Fanuc TP program (LS listing): 190220_hosenrohr_oV.ls

/PROG  190220_hosenrohr_oV
/ATTR
COMMENT	= "19-02-22 10:03:29";
PROG_SIZE	= 0;
DEFAULT_GROUP	= 1, 1, *, *, *;
/APPL
    ARC Welding Equipment: 1, *, *, *, *;
/MN
   1:  CALL HOME_ALL;
   1:  UFRAME_NUM = 1;
   1:  UTOOL_NUM = 3;
   1:  COL GUARD ADJUST 150;
   1:  ! -- Layer/Ebene 1 -- !;
   1:  PR[91] = PR[90];
   1:  PR[GP1:91,1] = PR[GP1:90,1] + -0.454;
   1:  PR[GP1:91,2] = PR[GP1:90,2] + 0.328;
   1:  PR[GP1:91,3] = PR[GP1:90,3] + 0.915;
   1:  !Sicherheitspunkt!;
   1:  PR[92] = PR[91];
   1:  PR[92] = PR[GP1:92,3] + 50;
   1:J PR[92];
   1:  !Schweissanfang anfahren!;
   1:L PR[91] R[100]mm/sec CNT100;
   1:  CALL LASER_DRAHT_START;
   1:  PR[GP1:91,1] = PR[GP1:90,1] + -4.023;
   1:  PR[GP1:91,2] = PR[GP1:90,2] + 1.652;
   1:L PR[91] R[100]mm/sec CNT100;
   1:  PR[GP1:91,1] = PR[GP1:90,1] + -5.839;
   1:  PR[GP1:91,2] = PR[GP1:90,2] + 4.932;
   1:L PR[91] R[100]mm/sec CNT100;
   1:  PR[GP1:91,1] = PR[GP1:90,1] + -9.924;
   1:  PR[GP1:91,2] = PR[GP1:90,2] + 16.574;
   1:L PR[91] R[100]mm/sec CNT100;
   1:  PR[GP1:91,1] = PR[GP1:90,1] + -10.007;
   1:  PR[GP1:91,2] = PR[GP1:90,2] + 16.909;
   1:L PR[91] R[100]mm/sec CNT100;
   1:  PR[GP1:91,1] = PR[GP1:90,1] + -10.104;
   1:  PR[GP1:91,2] = PR[GP1:90,2] + 17.121;
   1:L PR[91] R[100]mm/sec CNT100;
   1:  PR[GP1:91,1] = PR[GP1:90,1] + -18.076;
   1:  PR[GP1:91,2] = PR[GP1:90,2] + 26.372;
   1:L PR[91] R[100]mm/sec CNT100;
   1:  PR[GP1:91,1] = PR[GP1:90,1] + -18.276;
   1:  PR[GP1:91,2] = PR[GP1:90,2] + 26.653;
   1:L PR[91] R[100]mm/sec CNT100;
   1:  PR[GP1:91,1] = PR[GP1:90,1] + -18.444;
   1:  PR[GP1:91,2] = PR[GP1:90,2] + 26.815;
   1:L PR[91] R[100]mm/sec CNT100;
   1:  PR[GP1:91,1] = PR[GP1:90,1] + -29.237;
   1:  PR[GP1:91,2] = PR[GP1:90,2] + 32.512;
   1:L PR[91] R[100]mm/sec CNT100;
   1:  PR[GP1:91,1] = PR[GP1:90,1] + -29.526;
   1:  PR[GP1:91,2] = PR[GP1:90,2] + 32.701;
   1:L PR[91] R[100]mm/sec CNT100;
   1:  PR[GP1:91,1] = PR[GP1:90,1] + -29.741;
   1:  PR[GP1:91,2] = PR[GP1:90,2] + 32.790;
   1:L PR[91] R[100]mm/sec CNT100;
   1:  PR[GP1:91,1] = PR[GP1:90,1] + -41.876;
   1:  PR[GP1:91,2] = PR[GP1:90,2] + 34.153;
   1:L PR[91] R[100]mm/sec CNT100;
   1:  PR[GP1:91,1] = PR[GP1:90,1] + -42.214;
   1:  PR[GP1:91,2] = PR[GP1:90,2] + 34.223;
   1:L PR[91] R[100]mm/sec CNT100;
   1:  PR[GP1:91,1] = PR[GP1:90,1] + -42.447;
   1:  PR[GP1:91,2] = PR[GP1:90,2] + 34.227;
   1:L PR[91] R[100]mm/sec CNT100;
   1:  PR[GP1:91,1] = PR[GP1:90,1] + -54.241;
   1:  PR[GP1:91,2] = PR[GP1:90,2] + 31.064;
   1:L PR[91] R[100]mm/sec CNT100;
   1:  PR[GP1:91,1] = PR[GP1:90,1] + -54.581;
   1:  PR[GP1:91,2] = PR[GP1:90,2] + 31.006;
   1:L PR[91] R[100]mm/sec CNT100;
   1:  PR[GP1:91,1] = PR[GP1:90,1] + -54.799;
   1:  PR[GP1:91,2] = PR[GP1:90,2] + 30.925;
   1:L PR[91] R[100]mm/sec CNT100;
   1:  PR[GP1:91,1] = PR[GP1:90,1] + -64.619;
   1:  PR[GP1:91,2] = PR[GP1:90,2] + 23.675;
   1:L PR[91] R[100]mm/sec CNT100;
   1:  PR[GP1:91,1] = PR[GP1:90,1] + -64.915;
   1:  PR[GP1:91,2] = PR[GP1:90,2] + 23.497;
   1:L PR[91] R[100]mm/sec CNT100;
   1:  PR[GP1:91,1] = PR[GP1:90,1] + -65.088;
   1:  PR[GP1:91,2] = PR[GP1:90,2] + 23.342;
   1:L PR[91] R[100]mm/sec CNT100;
   1:  PR[GP1:91,1] = PR[GP1:90,1] + -71.586;
   1:  PR[GP1:91,2] = PR[GP1:90,2] + 12.999;
   1:L PR[91] R[100]mm/sec CNT100;
   1:  PR[GP1:91,1] = PR[GP1:90,1] + -71.796;
   1:  PR[GP1:91,2] = PR[GP1:90,2] + 12.725;
   1:L PR[91] R[100]mm/sec CNT100;
   1:  PR[GP1:91,1] = PR[GP1:90,1] + -71.901;
   1:  PR[GP1:91,2] = PR[GP1:90,2] + 12.518;
   1:L PR[91] R[100]mm/sec CNT100;
   1:  PR[GP1:91,1] = PR[GP1:90,1] + -74.171;
   1:  PR[GP1:91,2] = PR[GP1:90,2] + 0.520;
   1:L PR[91] R[100]mm/sec CNT100;
   1:  PR[GP1:91,1] = PR[GP1:90,1] + -74.266;
   1:  PR[GP1:91,2] = PR[GP1:90,2] + 0.188;
   1:L PR[91] R[100]mm/sec CNT100;
   1:  PR[GP1:91,1] = PR[GP1:90,1] + -74.288;
   1:  PR[GP1:91,2] = PR[GP1:90,2] + -0.044;
   1:L PR[91] R[100]mm/sec CNT100;
   1:  PR[GP1:91,1] = PR[GP1:90,1] + -72.018;
   1:  PR[GP1:91,2] = PR[GP1:90,2] + -12.041;
   1:L PR[91] R[100]mm/sec CNT100;
   1:  PR[GP1:91,1] = PR[GP1:90,1] + -71.986;
   1:  PR[GP1:91,2] = PR[GP1:90,2] + -12.385;
   1:L PR[91] R[100]mm/sec CNT100;
   1:  PR[GP1:91,1] = PR[GP1:90,1] + -71.914;
   1:  PR[GP1:91,2] = PR[GP1:90,2] + -12.636;
   1:L PR[91] R[100]mm/sec CNT100;
   1:  PR[GP1:91,1] = PR[GP1:90,1] + -71.783;
   1:  PR[GP1:91,2] = PR[GP1:90,2] + -12.894;
   1:L PR[91] R[100]mm/sec CNT100;
   1:  PR[GP1:91,1] = PR[GP1:90,1] + -65.286;
   1:  PR[GP1:91,2] = PR[GP1:90,2] + -23.237;
   1:L PR[91] R[100]mm/sec CNT100;
   1:  PR[GP1:91,1] = PR[GP1:90,1] + -65.109;
   1:  PR[GP1:91,2] = PR[GP1:90,2] + -23.467;
   1:L PR[91] R[100]mm/sec CNT100;
   1:  PR[GP1:91,1] = PR[GP1:90,1] + -64.894;
   1:  PR[GP1:91,2] = PR[GP1:90,2] + -23.659;
   1:L PR[91] R[100]mm/sec CNT100;
   1:  PR[GP1:91,1] = PR[GP1:90,1] + -55.074;
   1:  PR[GP1:91,2] = PR[GP1:90,2] + -30.910;
   1:L PR[91] R[100]mm/sec CNT100;
   1:  PR[GP1:91,1] = PR[GP1:90,1] + -54.826;
   1:  PR[GP1:91,2] = PR[GP1:90,2] + -31.059;
   1:L PR[91] R[100]mm/sec CNT100;
   1:  PR[GP1:91,1] = PR[GP1:90,1] + -54.555;
   1:  PR[GP1:91,2] = PR[GP1:90,2] + -31.160;
   1:L PR[91] R[100]mm/sec CNT100;
   1:  PR[GP1:91,1] = PR[GP1:90,1] + -42.760;
   1:  PR[GP1:91,2] = PR[GP1:90,2] + -34.323;
   1:L PR[91] R[100]mm/sec CNT100;
   1:  PR[GP1:91,1] = PR[GP1:90,1] + -42.475;
   1:  PR[GP1:91,2] = PR[GP1:90,2] + -34.372;
   1:L PR[91] R[100]mm/sec CNT100;
   1:  PR[GP1:91,1] = PR[GP1:90,1] + -42.186;
   1:  PR[GP1:91,2] = PR[GP1:90,2] + -34.367;
   1:L PR[91] R[100]mm/sec CNT100;
   1:  PR[GP1:91,1] = PR[GP1:90,1] + -30.051;
   1:  PR[GP1:91,2] = PR[GP1:90,2] + -33.004;
   1:L PR[91] R[100]mm/sec CNT100;
   1:  PR[GP1:91,1] = PR[GP1:90,1] + -29.768;
   1:  PR[GP1:91,2] = PR[GP1:90,2] + -32.945;
   1:L PR[91] R[100]mm/sec CNT100;
   1:  PR[GP1:91,1] = PR[GP1:90,1] + -29.500;
   1:  PR[GP1:91,2] = PR[GP1:90,2] + -32.835;
   1:L PR[91] R[100]mm/sec CNT100;
   1:  PR[GP1:91,1] = PR[GP1:90,1] + -18.706;
   1:  PR[GP1:91,2] = PR[GP1:90,2] + -27.137;
   1:L PR[91] R[100]mm/sec CNT100;
   1:  PR[GP1:91,1] = PR[GP1:90,1] + -18.464;
   1:  PR[GP1:91,2] = PR[GP1:90,2] + -26.978;
   1:L PR[91] R[100]mm/sec CNT100;
   1:  PR[GP1:91,1] = PR[GP1:90,1] + -18.256;
   1:  PR[GP1:91,2] = PR[GP1:90,2] + -26.778;
   1:L PR[91] R[100]mm/sec CNT100;
   1:  PR[GP1:91,1] = PR[GP1:90,1] + -10.284;
   1:  PR[GP1:91,2] = PR[GP1:90,2] + -17.526;
   1:L PR[91] R[100]mm/sec CNT100;
   1:  PR[GP1:91,1] = PR[GP1:90,1] + -10.116;
   1:  PR[GP1:91,2] = PR[GP1:90,2] + -17.290;
   1:L PR[91] R[100]mm/sec CNT100;
   1:  PR[GP1:91,1] = PR[GP1:90,1] + -9.995;
   1:  PR[GP1:91,2] = PR[GP1:90,2] + -17.028;
   1:L PR[91] R[100]mm/sec CNT100;
   1:  PR[GP1:91,1] = PR[GP1:90,1] + -5.955;
   1:  PR[GP1:91,2] = PR[GP1:90,2] + -5.512;
   1:L PR[91] R[100]mm/sec CNT100;
   1:  PR[GP1:91,1] = PR[GP1:90,1] + -5.853;
   1:  PR[GP1:91,2] = PR[GP1:90,2] + -5.100;
   1:L PR[91] R[100]mm/sec CNT100;
   1:  PR[GP1:91,1] = PR[GP1:90,1] + -4.023;
   1:  PR[GP1:91,2] = PR[GP1:90,2] + -1.796;
   1:L PR[91] R[100]mm/sec CNT100;
   1:  PR[GP1:91,1] = PR[GP1:90,1] + -0.454;
   1:  PR[GP1:91,2] = PR[GP1:90,2] + -0.472;
   1:L PR[91] R[100]mm/sec CNT100;
   1:  PR[GP1:91,1] = PR[GP1:90,1] + 0.667;
   1:L PR[91] R[100]mm/sec CNT100;
   1:  PR[GP1:91,1] = PR[GP1:90,1] + 4.237;
   1:  PR[GP1:91,2] = PR[GP1:90,2] + -1.796;
   1:L PR[91] R[100]mm/sec CNT100;
   1:  PR[GP1:91,1] = PR[GP1:90,1] + 6.052;
   1:  PR[GP1:91,2] = PR[GP1:90,2] + -5.076;
   1:L PR[91] R[100]mm/sec CNT100;
   1:  PR[GP1:91,1] = PR[GP1:90,1] + 10.137;
   1:  PR[GP1:91,2] = PR[GP1:90,2] + -16.718;
   1:L PR[91] R[100]mm/sec CNT100;
   1:  PR[GP1:91,1] = PR[GP1:90,1] + 10.221;
   1:  PR[GP1:91,2] = PR[GP1:90,2] + -17.053;
   1:L PR[91] R[100]mm/sec CNT100;
   1:  PR[GP1:91,1] = PR[GP1:90,1] + 10.318;
   1:  PR[GP1:91,2] = PR[GP1:90,2] + -17.265;
   1:L PR[91] R[100]mm/sec CNT100;
   1:  PR[GP1:91,1] = PR[GP1:90,1] + 18.289;
   1:  PR[GP1:91,2] = PR[GP1:90,2] + -26.516;
   1:L PR[91] R[100]mm/sec CNT100;
   1:  PR[GP1:91,1] = PR[GP1:90,1] + 18.489;
   1:  PR[GP1:91,2] = PR[GP1:90,2] + -26.797;
   1:L PR[91] R[100]mm/sec CNT100;
   1:  PR[GP1:91,1] = PR[GP1:90,1] + 18.657;
   1:  PR[GP1:91,2] = PR[GP1:90,2] + -26.959;
   1:L PR[91] R[100]mm/sec CNT100;
   1:  PR[GP1:91,1] = PR[GP1:90,1] + 29.451;
   1:  PR[GP1:91,2] = PR[GP1:90,2] + -32.656;
   1:L PR[91] R[100]mm/sec CNT100;
   1:  PR[GP1:91,1] = PR[GP1:90,1] + 29.740;
   1:  PR[GP1:91,2] = PR[GP1:90,2] + -32.845;
   1:L PR[91] R[100]mm/sec CNT100;
   1:  PR[GP1:91,1] = PR[GP1:90,1] + 29.955;
   1:  PR[GP1:91,2] = PR[GP1:90,2] + -32.934;
   1:L PR[91] R[100]mm/sec CNT100;
   1:  PR[GP1:91,1] = PR[GP1:90,1] + 42.089;
   1:  PR[GP1:91,2] = PR[GP1:90,2] + -34.297;
   1:L PR[91] R[100]mm/sec CNT100;
   1:  PR[GP1:91,1] = PR[GP1:90,1] + 42.427;
   1:  PR[GP1:91,2] = PR[GP1:90,2] + -34.367;
   1:L PR[91] R[100]mm/sec CNT100;
   1:  PR[GP1:91,1] = PR[GP1:90,1] + 42.660;
   1:  PR[GP1:91,2] = PR[GP1:90,2] + -34.371;
   1:L PR[91] R[100]mm/sec CNT100;
   1:  PR[GP1:91,1] = PR[GP1:90,1] + 54.454;
   1:  PR[GP1:91,2] = PR[GP1:90,2] + -31.208;
   1:L PR[91] R[100]mm/sec CNT100;
   1:  PR[GP1:91,1] = PR[GP1:90,1] + 54.794;
   1:  PR[GP1:91,2] = PR[GP1:90,2] + -31.150;
   1:L PR[91] R[100]mm/sec CNT100;
   1:  PR[GP1:91,1] = PR[GP1:90,1] + 55.013;
   1:  PR[GP1:91,2] = PR[GP1:90,2] + -31.069;
   1:L PR[91] R[100]mm/sec CNT100;
   1:  PR[GP1:91,1] = PR[GP1:90,1] + 64.832;
   1:  PR[GP1:91,2] = PR[GP1:90,2] + -23.819;
   1:L PR[91] R[100]mm/sec CNT100;
   1:  PR[GP1:91,1] = PR[GP1:90,1] + 65.128;
   1:  PR[GP1:91,2] = PR[GP1:90,2] + -23.641;
   1:L PR[91] R[100]mm/sec CNT100;
   1:  PR[GP1:91,1] = PR[GP1:90,1] + 65.302;
   1:  PR[GP1:91,2] = PR[GP1:90,2] + -23.486;
   1:L PR[91] R[100]mm/sec CNT100;
   1:  PR[GP1:91,1] = PR[GP1:90,1] + 71.799;
   1:  PR[GP1:91,2] = PR[GP1:90,2] + -13.143;
   1:L PR[91] R[100]mm/sec CNT100;
   1:  PR[GP1:91,1] = PR[GP1:90,1] + 72.009;
   1:  PR[GP1:91,2] = PR[GP1:90,2] + -12.869;
   1:L PR[91] R[100]mm/sec CNT100;
   1:  PR[GP1:91,1] = PR[GP1:90,1] + 72.114;
   1:  PR[GP1:91,2] = PR[GP1:90,2] + -12.661;
   1:L PR[91] R[100]mm/sec CNT100;
   1:  PR[GP1:91,1] = PR[GP1:90,1] + 74.384;
   1:  PR[GP1:91,2] = PR[GP1:90,2] + -0.664;
   1:L PR[91] R[100]mm/sec CNT100;
   1:  PR[GP1:91,1] = PR[GP1:90,1] + 74.480;
   1:  PR[GP1:91,2] = PR[GP1:90,2] + -0.332;
   1:L PR[91] R[100]mm/sec CNT100;
   1:  PR[GP1:91,1] = PR[GP1:90,1] + 74.501;
   1:  PR[GP1:91,2] = PR[GP1:90,2] + -0.100;
   1:L PR[91] R[100]mm/sec CNT100;
   1:  PR[GP1:91,1] = PR[GP1:90,1] + 72.231;
   1:  PR[GP1:91,2] = PR[GP1:90,2] + 11.897;
   1:L PR[91] R[100]mm/sec CNT100;
   1:  PR[GP1:91,1] = PR[GP1:90,1] + 72.199;
   1:  PR[GP1:91,2] = PR[GP1:90,2] + 12.241;
   1:L PR[91] R[100]mm/sec CNT100;
   1:  PR[GP1:91,1] = PR[GP1:90,1] + 72.127;
   1:  PR[GP1:91,2] = PR[GP1:90,2] + 12.492;
   1:L PR[91] R[100]mm/sec CNT100;
   1:  PR[GP1:91,1] = PR[GP1:90,1] + 71.996;
   1:  PR[GP1:91,2] = PR[GP1:90,2] + 12.750;
   1:L PR[91] R[100]mm/sec CNT100;
   1:  PR[GP1:91,1] = PR[GP1:90,1] + 65.499;
   1:  PR[GP1:91,2] = PR[GP1:90,2] + 23.093;
   1:L PR[91] R[100]mm/sec CNT100;
   1:  PR[GP1:91,1] = PR[GP1:90,1] + 65.323;
   1:  PR[GP1:91,2] = PR[GP1:90,2] + 23.323;
   1:L PR[91] R[100]mm/sec CNT100;
   1:  PR[GP1:91,1] = PR[GP1:90,1] + 65.107;
   1:  PR[GP1:91,2] = PR[GP1:90,2] + 23.515;
   1:L PR[91] R[100]mm/sec CNT100;
   1:  PR[GP1:91,1] = PR[GP1:90,1] + 55.287;
   1:  PR[GP1:91,2] = PR[GP1:90,2] + 30.766;
   1:L PR[91] R[100]mm/sec CNT100;
   1:  PR[GP1:91,1] = PR[GP1:90,1] + 55.039;
   1:  PR[GP1:91,2] = PR[GP1:90,2] + 30.915;
   1:L PR[91] R[100]mm/sec CNT100;
   1:  PR[GP1:91,1] = PR[GP1:90,1] + 54.768;
   1:  PR[GP1:91,2] = PR[GP1:90,2] + 31.016;
   1:L PR[91] R[100]mm/sec CNT100;
   1:  PR[GP1:91,1] = PR[GP1:90,1] + 42.973;
   1:  PR[GP1:91,2] = PR[GP1:90,2] + 34.179;
   1:L PR[91] R[100]mm/sec CNT100;
   1:  PR[GP1:91,1] = PR[GP1:90,1] + 42.688;
   1:  PR[GP1:91,2] = PR[GP1:90,2] + 34.228;
   1:L PR[91] R[100]mm/sec CNT100;
   1:  PR[GP1:91,1] = PR[GP1:90,1] + 42.399;
   1:  PR[GP1:91,2] = PR[GP1:90,2] + 34.223;
   1:L PR[91] R[100]mm/sec CNT100;
   1:  PR[GP1:91,1] = PR[GP1:90,1] + 30.264;
   1:  PR[GP1:91,2] = PR[GP1:90,2] + 32.860;
   1:L PR[91] R[100]mm/sec CNT100;
   1:  PR[GP1:91,1] = PR[GP1:90,1] + 29.981;
   1:  PR[GP1:91,2] = PR[GP1:90,2] + 32.801;
   1:L PR[91] R[100]mm/sec CNT100;
   1:  PR[GP1:91,1] = PR[GP1:90,1] + 29.714;
   1:  PR[GP1:91,2] = PR[GP1:90,2] + 32.691;
   1:L PR[91] R[100]mm/sec CNT100;
   1:  PR[GP1:91,1] = PR[GP1:90,1] + 18.920;
   1:  PR[GP1:91,2] = PR[GP1:90,2] + 26.993;
   1:L PR[91] R[100]mm/sec CNT100;
   1:  PR[GP1:91,1] = PR[GP1:90,1] + 18.678;
   1:  PR[GP1:91,2] = PR[GP1:90,2] + 26.834;
   1:L PR[91] R[100]mm/sec CNT100;
   1:  PR[GP1:91,1] = PR[GP1:90,1] + 18.469;
   1:  PR[GP1:91,2] = PR[GP1:90,2] + 26.634;
   1:L PR[91] R[100]mm/sec CNT100;
   1:  PR[GP1:91,1] = PR[GP1:90,1] + 10.497;
   1:  PR[GP1:91,2] = PR[GP1:90,2] + 17.382;
   1:L PR[91] R[100]mm/sec CNT100;
   1:  PR[GP1:91,1] = PR[GP1:90,1] + 10.330;
   1:  PR[GP1:91,2] = PR[GP1:90,2] + 17.146;
   1:L PR[91] R[100]mm/sec CNT100;
   1:  PR[GP1:91,1] = PR[GP1:90,1] + 10.209;
   1:  PR[GP1:91,2] = PR[GP1:90,2] + 16.884;
   1:L PR[91] R[100]mm/sec CNT100;
   1:  PR[GP1:91,1] = PR[GP1:90,1] + 6.168;
   1:  PR[GP1:91,2] = PR[GP1:90,2] + 5.368;
   1:L PR[91] R[100]mm/sec CNT100;
   1:  PR[GP1:91,1] = PR[GP1:90,1] + 6.066;
   1:  PR[GP1:91,2] = PR[GP1:90,2] + 4.956;
   1:L PR[91] R[100]mm/sec CNT100;
   1:  PR[GP1:91,1] = PR[GP1:90,1] + 4.237;
   1:  PR[GP1:91,2] = PR[GP1:90,2] + 1.652;
   1:L PR[91] R[100]mm/sec CNT100;
   1:  PR[GP1:91,1] = PR[GP1:90,1] + 0.667;
   1:  PR[GP1:91,2] = PR[GP1:90,2] + 0.328;
   1:L PR[91] R[100]mm/sec CNT100;
   1:  PR[GP1:91,1] = PR[GP1:90,1] + -0.454;
   1:L PR[91] R[100]mm/sec CNT100;
   1:  ! -- Layer/Ebene 2 -- !;
   1:  PR[91] = PR[90];
   1:  PR[GP1:91,1] = PR[GP1:90,1] + -4.023;
   1:  PR[GP1:91,2] = PR[GP1:90,2] + 1.652;
   1:  PR[GP1:91,3] = PR[GP1:90,3] + 1.525;
   1:L PR[91] R[100]mm/sec CNT100;
   1:  PR[GP1:91,1] = PR[GP1:90,1] + -5.839;
   1:  PR[GP1:91,2] = PR[GP1:90,2] + 4.932;
   1:L PR[91] R[100]mm/sec CNT100;
   1:  PR[GP1:91,1] = PR[GP1:90,1] + -9.513;
   1:  PR[GP1:91,2] = PR[GP1:90,2] + 15.405;
   1:L PR[91] R[100]mm/sec CNT100;
   1:  PR[GP1:91,1] = PR[GP1:90,1] + -9.747;
   1:  PR[GP1:91,2] = PR[GP1:90,2] + 16.344;
   1:L PR[91] R[100]mm/sec CNT100;
   1:  PR[GP1:91,1] = PR[GP1:90,1] + -10.105;
   1:  PR[GP1:91,2] = PR[GP1:90,2] + 17.121;
   1:L PR[91] R[100]mm/sec CNT100;
   1:  PR[GP1:91,1] = PR[GP1:90,1] + -17.267;
   1:  PR[GP1:91,2] = PR[GP1:90,2] + 25.433;
   1:L PR[91] R[100]mm/sec CNT100;
   1:  PR[GP1:91,1] = PR[GP1:90,1] + -17.828;
   1:  PR[GP1:91,2] = PR[GP1:90,2] + 26.222;
   1:L PR[91] R[100]mm/sec CNT100;
   1:  PR[GP1:91,1] = PR[GP1:90,1] + -18.444;
   1:  PR[GP1:91,2] = PR[GP1:90,2] + 26.815;
   1:L PR[91] R[100]mm/sec CNT100;
   1:  PR[GP1:91,1] = PR[GP1:90,1] + -28.141;
   1:  PR[GP1:91,2] = PR[GP1:90,2] + 31.934;
   1:L PR[91] R[100]mm/sec CNT100;
   1:  PR[GP1:91,1] = PR[GP1:90,1] + -28.952;
   1:  PR[GP1:91,2] = PR[GP1:90,2] + 32.464;
   1:L PR[91] R[100]mm/sec CNT100;
   1:  PR[GP1:91,1] = PR[GP1:90,1] + -29.742;
   1:  PR[GP1:91,2] = PR[GP1:90,2] + 32.791;
   1:L PR[91] R[100]mm/sec CNT100;
   1:  PR[GP1:91,1] = PR[GP1:90,1] + -40.644;
   1:  PR[GP1:91,2] = PR[GP1:90,2] + 34.015;
   1:L PR[91] R[100]mm/sec CNT100;
   1:  PR[GP1:91,1] = PR[GP1:90,1] + -41.592;
   1:  PR[GP1:91,2] = PR[GP1:90,2] + 34.212;
   1:L PR[91] R[100]mm/sec CNT100;
   1:  PR[GP1:91,1] = PR[GP1:90,1] + -42.447;
   1:  PR[GP1:91,2] = PR[GP1:90,2] + 34.227;
   1:L PR[91] R[100]mm/sec CNT100;
   1:  PR[GP1:91,1] = PR[GP1:90,1] + -53.043;
   1:  PR[GP1:91,2] = PR[GP1:90,2] + 31.385;
   1:L PR[91] R[100]mm/sec CNT100;
   1:  PR[GP1:91,1] = PR[GP1:90,1] + -53.998;
   1:  PR[GP1:91,2] = PR[GP1:90,2] + 31.223;
   1:L PR[91] R[100]mm/sec CNT100;
   1:  PR[GP1:91,1] = PR[GP1:90,1] + -54.800;
   1:  PR[GP1:91,2] = PR[GP1:90,2] + 30.925;
   1:L PR[91] R[100]mm/sec CNT100;
   1:  PR[GP1:91,1] = PR[GP1:90,1] + -63.622;
   1:  PR[GP1:91,2] = PR[GP1:90,2] + 24.411;
   1:L PR[91] R[100]mm/sec CNT100;
   1:  PR[GP1:91,1] = PR[GP1:90,1] + -64.451;
   1:  PR[GP1:91,2] = PR[GP1:90,2] + 23.911;
   1:L PR[91] R[100]mm/sec CNT100;
   1:  PR[GP1:91,1] = PR[GP1:90,1] + -65.089;
   1:  PR[GP1:91,2] = PR[GP1:90,2] + 23.341;
   1:L PR[91] R[100]mm/sec CNT100;
   1:  PR[GP1:91,1] = PR[GP1:90,1] + -70.926;
   1:  PR[GP1:91,2] = PR[GP1:90,2] + 14.049;
   1:L PR[91] R[100]mm/sec CNT100;
   1:  PR[GP1:91,1] = PR[GP1:90,1] + -71.515;
   1:  PR[GP1:91,2] = PR[GP1:90,2] + 13.281;
   1:L PR[91] R[100]mm/sec CNT100;
   1:  PR[GP1:91,1] = PR[GP1:90,1] + -71.901;
   1:  PR[GP1:91,2] = PR[GP1:90,2] + 12.517;
   1:L PR[91] R[100]mm/sec CNT100;
   1:  PR[GP1:91,1] = PR[GP1:90,1] + -73.940;
   1:  PR[GP1:91,2] = PR[GP1:90,2] + 1.738;
   1:L PR[91] R[100]mm/sec CNT100;
   1:  PR[GP1:91,1] = PR[GP1:90,1] + -74.208;
   1:  PR[GP1:91,2] = PR[GP1:90,2] + 0.808;
   1:L PR[91] R[100]mm/sec CNT100;
   1:  PR[GP1:91,1] = PR[GP1:90,1] + -74.288;
   1:  PR[GP1:91,2] = PR[GP1:90,2] + -0.044;
   1:L PR[91] R[100]mm/sec CNT100;
   1:  PR[GP1:91,1] = PR[GP1:90,1] + -72.249;
   1:  PR[GP1:91,2] = PR[GP1:90,2] + -10.823;
   1:L PR[91] R[100]mm/sec CNT100;
   1:  PR[GP1:91,1] = PR[GP1:90,1] + -72.158;
   1:  PR[GP1:91,2] = PR[GP1:90,2] + -11.787;
   1:L PR[91] R[100]mm/sec CNT100;
   1:  PR[GP1:91,1] = PR[GP1:90,1] + -71.914;
   1:  PR[GP1:91,2] = PR[GP1:90,2] + -12.636;
   1:L PR[91] R[100]mm/sec CNT100;
   1:  PR[GP1:91,1] = PR[GP1:90,1] + -71.503;
   1:  PR[GP1:91,2] = PR[GP1:90,2] + -13.450;
   1:L PR[91] R[100]mm/sec CNT100;
   1:  PR[GP1:91,1] = PR[GP1:90,1] + -65.665;
   1:  PR[GP1:91,2] = PR[GP1:90,2] + -22.742;
   1:L PR[91] R[100]mm/sec CNT100;
   1:  PR[GP1:91,1] = PR[GP1:90,1] + -65.110;
   1:  PR[GP1:91,2] = PR[GP1:90,2] + -23.466;
   1:L PR[91] R[100]mm/sec CNT100;
   1:  PR[GP1:91,1] = PR[GP1:90,1] + -64.430;
   1:  PR[GP1:91,2] = PR[GP1:90,2] + -24.074;
   1:L PR[91] R[100]mm/sec CNT100;
   1:  PR[GP1:91,1] = PR[GP1:90,1] + -55.607;
   1:  PR[GP1:91,2] = PR[GP1:90,2] + -30.588;
   1:L PR[91] R[100]mm/sec CNT100;
   1:  PR[GP1:91,1] = PR[GP1:90,1] + -54.826;
   1:  PR[GP1:91,2] = PR[GP1:90,2] + -31.059;
   1:L PR[91] R[100]mm/sec CNT100;
   1:  PR[GP1:91,1] = PR[GP1:90,1] + -53.971;
   1:  PR[GP1:91,2] = PR[GP1:90,2] + -31.376;
   1:L PR[91] R[100]mm/sec CNT100;
   1:  PR[GP1:91,1] = PR[GP1:90,1] + -43.375;
   1:  PR[GP1:91,2] = PR[GP1:90,2] + -34.219;
   1:L PR[91] R[100]mm/sec CNT100;
   1:  PR[GP1:91,1] = PR[GP1:90,1] + -42.476;
   1:  PR[GP1:91,2] = PR[GP1:90,2] + -34.372;
   1:L PR[91] R[100]mm/sec CNT100;
   1:  PR[GP1:91,1] = PR[GP1:90,1] + -41.564;
   1:  PR[GP1:91,2] = PR[GP1:90,2] + -34.355;
   1:L PR[91] R[100]mm/sec CNT100;
   1:  PR[GP1:91,1] = PR[GP1:90,1] + -30.661;
   1:  PR[GP1:91,2] = PR[GP1:90,2] + -33.131;
   1:L PR[91] R[100]mm/sec CNT100;
   1:  PR[GP1:91,1] = PR[GP1:90,1] + -29.768;
   1:  PR[GP1:91,2] = PR[GP1:90,2] + -32.945;
   1:L PR[91] R[100]mm/sec CNT100;
   1:  PR[GP1:91,1] = PR[GP1:90,1] + -28.926;
   1:  PR[GP1:91,2] = PR[GP1:90,2] + -32.597;
   1:L PR[91] R[100]mm/sec CNT100;
   1:  PR[GP1:91,1] = PR[GP1:90,1] + -19.228;
   1:  PR[GP1:91,2] = PR[GP1:90,2] + -27.478;
   1:L PR[91] R[100]mm/sec CNT100;
   1:  PR[GP1:91,1] = PR[GP1:90,1] + -18.465;
   1:  PR[GP1:91,2] = PR[GP1:90,2] + -26.979;
   1:L PR[91] R[100]mm/sec CNT100;
   1:  PR[GP1:91,1] = PR[GP1:90,1] + -17.807;
   1:  PR[GP1:91,2] = PR[GP1:90,2] + -26.346;
   1:L PR[91] R[100]mm/sec CNT100;
   1:  PR[GP1:91,1] = PR[GP1:90,1] + -10.645;
   1:  PR[GP1:91,2] = PR[GP1:90,2] + -18.034;
   1:L PR[91] R[100]mm/sec CNT100;
   1:  PR[GP1:91,1] = PR[GP1:90,1] + -10.117;
   1:  PR[GP1:91,2] = PR[GP1:90,2] + -17.291;
   1:L PR[91] R[100]mm/sec CNT100;
   1:  PR[GP1:91,1] = PR[GP1:90,1] + -9.736;
   1:  PR[GP1:91,2] = PR[GP1:90,2] + -16.462;
   1:L PR[91] R[100]mm/sec CNT100;
   1:  PR[GP1:91,1] = PR[GP1:90,1] + -6.106;
   1:  PR[GP1:91,2] = PR[GP1:90,2] + -6.117;
   1:L PR[91] R[100]mm/sec CNT100;
   1:  PR[GP1:91,1] = PR[GP1:90,1] + -5.853;
   1:  PR[GP1:91,2] = PR[GP1:90,2] + -5.100;
   1:L PR[91] R[100]mm/sec CNT100;
   1:  PR[GP1:91,1] = PR[GP1:90,1] + -4.023;
   1:  PR[GP1:91,2] = PR[GP1:90,2] + -1.796;
   1:L PR[91] R[100]mm/sec CNT100;
   1:  PR[GP1:91,1] = PR[GP1:90,1] + -0.454;
   1:  PR[GP1:91,2] = PR[GP1:90,2] + -0.472;
   1:L PR[91] R[100]mm/sec CNT100;
   1:  PR[GP1:91,1] = PR[GP1:90,1] + 0.667;
   1:L PR[91] R[100]mm/sec CNT100;
   1:  PR[GP1:91,1] = PR[GP1:90,1] + 4.237;
   1:  PR[GP1:91,2] = PR[GP1:90,2] + -1.796;
   1:L PR[91] R[100]mm/sec CNT100;
   1:  PR[GP1:91,1] = PR[GP1:90,1] + 6.052;
   1:  PR[GP1:91,2] = PR[GP1:90,2] + -5.076;
   1:L PR[91] R[100]mm/sec CNT100;
   1:  PR[GP1:91,1] = PR[GP1:90,1] + 9.727;
   1:  PR[GP1:91,2] = PR[GP1:90,2] + -15.549;
   1:L PR[91] R[100]mm/sec CNT100;
   1:  PR[GP1:91,1] = PR[GP1:90,1] + 9.961;
   1:  PR[GP1:91,2] = PR[GP1:90,2] + -16.488;
   1:L PR[91] R[100]mm/sec CNT100;
   1:  PR[GP1:91,1] = PR[GP1:90,1] + 10.318;
   1:  PR[GP1:91,2] = PR[GP1:90,2] + -17.265;
   1:L PR[91] R[100]mm/sec CNT100;
   1:  PR[GP1:91,1] = PR[GP1:90,1] + 17.480;
   1:  PR[GP1:91,2] = PR[GP1:90,2] + -25.577;
   1:L PR[91] R[100]mm/sec CNT100;
   1:  PR[GP1:91,1] = PR[GP1:90,1] + 18.041;
   1:  PR[GP1:91,2] = PR[GP1:90,2] + -26.366;
   1:L PR[91] R[100]mm/sec CNT100;
   1:  PR[GP1:91,1] = PR[GP1:90,1] + 18.657;
   1:  PR[GP1:91,2] = PR[GP1:90,2] + -26.959;
   1:L PR[91] R[100]mm/sec CNT100;
   1:  PR[GP1:91,1] = PR[GP1:90,1] + 28.355;
   1:  PR[GP1:91,2] = PR[GP1:90,2] + -32.078;
   1:L PR[91] R[100]mm/sec CNT100;
   1:  PR[GP1:91,1] = PR[GP1:90,1] + 29.165;
   1:  PR[GP1:91,2] = PR[GP1:90,2] + -32.608;
   1:L PR[91] R[100]mm/sec CNT100;
   1:  PR[GP1:91,1] = PR[GP1:90,1] + 29.955;
   1:  PR[GP1:91,2] = PR[GP1:90,2] + -32.934;
   1:L PR[91] R[100]mm/sec CNT100;
   1:  PR[GP1:91,1] = PR[GP1:90,1] + 40.857;
   1:  PR[GP1:91,2] = PR[GP1:90,2] + -34.159;
   1:L PR[91] R[100]mm/sec CNT100;
   1:  PR[GP1:91,1] = PR[GP1:90,1] + 41.805;
   1:  PR[GP1:91,2] = PR[GP1:90,2] + -34.356;
   1:L PR[91] R[100]mm/sec CNT100;
   1:  PR[GP1:91,1] = PR[GP1:90,1] + 42.660;
   1:  PR[GP1:91,2] = PR[GP1:90,2] + -34.371;
   1:L PR[91] R[100]mm/sec CNT100;
   1:  PR[GP1:91,1] = PR[GP1:90,1] + 53.257;
   1:  PR[GP1:91,2] = PR[GP1:90,2] + -31.529;
   1:L PR[91] R[100]mm/sec CNT100;
   1:  PR[GP1:91,1] = PR[GP1:90,1] + 54.211;
   1:  PR[GP1:91,2] = PR[GP1:90,2] + -31.367;
   1:L PR[91] R[100]mm/sec CNT100;
   1:  PR[GP1:91,1] = PR[GP1:90,1] + 55.013;
   1:  PR[GP1:91,2] = PR[GP1:90,2] + -31.069;
   1:L PR[91] R[100]mm/sec CNT100;
   1:  PR[GP1:91,1] = PR[GP1:90,1] + 63.835;
   1:  PR[GP1:91,2] = PR[GP1:90,2] + -24.555;
   1:L PR[91] R[100]mm/sec CNT100;
   1:  PR[GP1:91,1] = PR[GP1:90,1] + 64.664;
   1:  PR[GP1:91,2] = PR[GP1:90,2] + -24.055;
   1:L PR[91] R[100]mm/sec CNT100;
   1:  PR[GP1:91,1] = PR[GP1:90,1] + 65.302;
   1:  PR[GP1:91,2] = PR[GP1:90,2] + -23.485;
   1:L PR[91] R[100]mm/sec CNT100;
   1:  PR[GP1:91,1] = PR[GP1:90,1] + 71.140;
   1:  PR[GP1:91,2] = PR[GP1:90,2] + -14.193;
   1:L PR[91] R[100]mm/sec CNT100;
   1:  PR[GP1:91,1] = PR[GP1:90,1] + 71.729;
   1:  PR[GP1:91,2] = PR[GP1:90,2] + -13.425;
   1:L PR[91] R[100]mm/sec CNT100;
   1:  PR[GP1:91,1] = PR[GP1:90,1] + 72.114;
   1:  PR[GP1:91,2] = PR[GP1:90,2] + -12.661;
   1:L PR[91] R[100]mm/sec CNT100;
   1:  PR[GP1:91,1] = PR[GP1:90,1] + 74.154;
   1:  PR[GP1:91,2] = PR[GP1:90,2] + -1.882;
   1:L PR[91] R[100]mm/sec CNT100;
   1:  PR[GP1:91,1] = PR[GP1:90,1] + 74.421;
   1:  PR[GP1:91,2] = PR[GP1:90,2] + -0.952;
   1:L PR[91] R[100]mm/sec CNT100;
   1:  PR[GP1:91,1] = PR[GP1:90,1] + 74.501;
   1:  PR[GP1:91,2] = PR[GP1:90,2] + -0.100;
   1:L PR[91] R[100]mm/sec CNT100;
   1:  PR[GP1:91,1] = PR[GP1:90,1] + 72.462;
   1:  PR[GP1:91,2] = PR[GP1:90,2] + 10.679;
   1:L PR[91] R[100]mm/sec CNT100;
   1:  PR[GP1:91,1] = PR[GP1:90,1] + 72.371;
   1:  PR[GP1:91,2] = PR[GP1:90,2] + 11.643;
   1:L PR[91] R[100]mm/sec CNT100;
   1:  PR[GP1:91,1] = PR[GP1:90,1] + 72.127;
   1:  PR[GP1:91,2] = PR[GP1:90,2] + 12.492;
   1:L PR[91] R[100]mm/sec CNT100;
   1:  PR[GP1:91,1] = PR[GP1:90,1] + 71.716;
   1:  PR[GP1:91,2] = PR[GP1:90,2] + 13.306;
   1:L PR[91] R[100]mm/sec CNT100;
   1:  PR[GP1:91,1] = PR[GP1:90,1] + 65.878;
   1:  PR[GP1:91,2] = PR[GP1:90,2] + 22.599;
   1:L PR[91] R[100]mm/sec CNT100;
   1:  PR[GP1:91,1] = PR[GP1:90,1] + 65.323;
   1:  PR[GP1:91,2] = PR[GP1:90,2] + 23.322;
   1:L PR[91] R[100]mm/sec CNT100;
   1:  PR[GP1:91,1] = PR[GP1:90,1] + 64.643;
   1:  PR[GP1:91,2] = PR[GP1:90,2] + 23.930;
   1:L PR[91] R[100]mm/sec CNT100;
   1:  PR[GP1:91,1] = PR[GP1:90,1] + 55.820;
   1:  PR[GP1:91,2] = PR[GP1:90,2] + 30.444;
   1:L PR[91] R[100]mm/sec CNT100;
   1:  PR[GP1:91,1] = PR[GP1:90,1] + 55.039;
   1:  PR[GP1:91,2] = PR[GP1:90,2] + 30.915;
   1:L PR[91] R[100]mm/sec CNT100;
   1:  PR[GP1:91,1] = PR[GP1:90,1] + 54.185;
   1:  PR[GP1:91,2] = PR[GP1:90,2] + 31.232;
   1:L PR[91] R[100]mm/sec CNT100;
   1:  PR[GP1:91,1] = PR[GP1:90,1] + 43.588;
   1:  PR[GP1:91,2] = PR[GP1:90,2] + 34.075;
   1:L PR[91] R[100]mm/sec CNT100;
   1:  PR[GP1:91,1] = PR[GP1:90,1] + 42.689;
   1:  PR[GP1:91,2] = PR[GP1:90,2] + 34.228;
   1:L PR[91] R[100]mm/sec CNT100;
   1:  PR[GP1:91,1] = PR[GP1:90,1] + 41.777;
   1:  PR[GP1:91,2] = PR[GP1:90,2] + 34.211;
   1:L PR[91] R[100]mm/sec CNT100;
   1:  PR[GP1:91,1] = PR[GP1:90,1] + 30.875;
   1:  PR[GP1:91,2] = PR[GP1:90,2] + 32.987;
   1:L PR[91] R[100]mm/sec CNT100;
   1:  PR[GP1:91,1] = PR[GP1:90,1] + 29.982;
   1:  PR[GP1:91,2] = PR[GP1:90,2] + 32.801;
   1:L PR[91] R[100]mm/sec CNT100;
   1:  PR[GP1:91,1] = PR[GP1:90,1] + 29.139;
   1:  PR[GP1:91,2] = PR[GP1:90,2] + 32.453;
   1:L PR[91] R[100]mm/sec CNT100;
   1:  PR[GP1:91,1] = PR[GP1:90,1] + 19.441;
   1:  PR[GP1:91,2] = PR[GP1:90,2] + 27.334;
   1:L PR[91] R[100]mm/sec CNT100;
   1:  PR[GP1:91,1] = PR[GP1:90,1] + 18.678;
   1:  PR[GP1:91,2] = PR[GP1:90,2] + 26.835;
   1:L PR[91] R[100]mm/sec CNT100;
   1:  PR[GP1:91,1] = PR[GP1:90,1] + 18.020;
   1:  PR[GP1:91,2] = PR[GP1:90,2] + 26.202;
   1:L PR[91] R[100]mm/sec CNT100;
   1:  PR[GP1:91,1] = PR[GP1:90,1] + 10.858;
   1:  PR[GP1:91,2] = PR[GP1:90,2] + 17.890;
   1:L PR[91] R[100]mm/sec CNT100;
   1:  PR[GP1:91,1] = PR[GP1:90,1] + 10.330;
   1:  PR[GP1:91,2] = PR[GP1:90,2] + 17.147;
   1:L PR[91] R[100]mm/sec CNT100;
   1:  PR[GP1:91,1] = PR[GP1:90,1] + 9.949;
   1:  PR[GP1:91,2] = PR[GP1:90,2] + 16.318;
   1:L PR[91] R[100]mm/sec CNT100;
   1:  PR[GP1:91,1] = PR[GP1:90,1] + 6.319;
   1:  PR[GP1:91,2] = PR[GP1:90,2] + 5.973;
   1:L PR[91] R[100]mm/sec CNT100;
   1:  PR[GP1:91,1] = PR[GP1:90,1] + 6.066;
   1:  PR[GP1:91,2] = PR[GP1:90,2] + 4.956;
   1:L PR[91] R[100]mm/sec CNT100;
   1:  PR[GP1:91,1] = PR[GP1:90,1] + 4.237;
   1:  PR[GP1:91,2] = PR[GP1:90,2] + 1.652;
   1:L PR[91] R[100]mm/sec CNT100;
   1:  PR[GP1:91,1] = PR[GP1:90,1] + 0.667;
   1:  PR[GP1:91,2] = PR[GP1:90,2] + 0.328;
   1:L PR[91] R[100]mm/sec CNT100;
   1:  PR[GP1:91,1] = PR[GP1:90,1] + -0.454;
   1:L PR[91] R[100]mm/sec CNT100;
   1:  ! -- Layer/Ebene 3 -- !;
   1:  PR[91] = PR[90];
   1:  PR[GP1:91,1] = PR[GP1:90,1] + -4.023;
   1:  PR[GP1:91,2] = PR[GP1:90,2] + 1.652;
   1:  PR[GP1:91,3] = PR[GP1:90,3] + 2.135;
   1:L PR[91] R[100]mm/sec CNT100;
   1:  PR[GP1:91,1] = PR[GP1:90,1] + -5.839;
   1:  PR[GP1:91,2] = PR[GP1:90,2] + 4.932;
   1:L PR[91] R[100]mm/sec CNT100;
   1:  PR[GP1:91,1] = PR[GP1:90,1] + -9.185;
   1:  PR[GP1:91,2] = PR[GP1:90,2] + 14.469;
   1:L PR[91] R[100]mm/sec CNT100;
   1:  PR[GP1:91,1] = PR[GP1:90,1] + -9.539;
   1:  PR[GP1:91,2] = PR[GP1:90,2] + 15.892;
   1:L PR[91] R[100]mm/sec CNT100;
   1:  PR[GP1:91,1] = PR[GP1:90,1] + -10.105;
   1:  PR[GP1:91,2] = PR[GP1:90,2] + 17.122;
   1:L PR[91] R[100]mm/sec CNT100;
   1:  PR[GP1:91,1] = PR[GP1:90,1] + -16.619;
   1:  PR[GP1:91,2] = PR[GP1:90,2] + 24.682;
   1:L PR[91] R[100]mm/sec CNT100;
   1:  PR[GP1:91,1] = PR[GP1:90,1] + -17.469;
   1:  PR[GP1:91,2] = PR[GP1:90,2] + 25.877;
   1:L PR[91] R[100]mm/sec CNT100;
   1:  PR[GP1:91,1] = PR[GP1:90,1] + -18.444;
   1:  PR[GP1:91,2] = PR[GP1:90,2] + 26.815;
   1:L PR[91] R[100]mm/sec CNT100;
   1:  PR[GP1:91,1] = PR[GP1:90,1] + -27.265;
   1:  PR[GP1:91,2] = PR[GP1:90,2] + 31.471;
   1:L PR[91] R[100]mm/sec CNT100;
   1:  PR[GP1:91,1] = PR[GP1:90,1] + -28.492;
   1:  PR[GP1:91,2] = PR[GP1:90,2] + 32.273;
   1:L PR[91] R[100]mm/sec CNT100;
   1:  PR[GP1:91,1] = PR[GP1:90,1] + -29.743;
   1:  PR[GP1:91,2] = PR[GP1:90,2] + 32.791;
   1:L PR[91] R[100]mm/sec CNT100;
   1:  PR[GP1:91,1] = PR[GP1:90,1] + -39.659;
   1:  PR[GP1:91,2] = PR[GP1:90,2] + 33.904;
   1:L PR[91] R[100]mm/sec CNT100;
   1:  PR[GP1:91,1] = PR[GP1:90,1] + -41.094;
   1:  PR[GP1:91,2] = PR[GP1:90,2] + 34.203;
   1:L PR[91] R[100]mm/sec CNT100;
   1:  PR[GP1:91,1] = PR[GP1:90,1] + -42.448;
   1:  PR[GP1:91,2] = PR[GP1:90,2] + 34.227;
   1:L PR[91] R[100]mm/sec CNT100;
   1:  PR[GP1:91,1] = PR[GP1:90,1] + -52.086;
   1:  PR[GP1:91,2] = PR[GP1:90,2] + 31.642;
   1:L PR[91] R[100]mm/sec CNT100;
   1:  PR[GP1:91,1] = PR[GP1:90,1] + -53.531;
   1:  PR[GP1:91,2] = PR[GP1:90,2] + 31.396;
   1:L PR[91] R[100]mm/sec CNT100;
   1:  PR[GP1:91,1] = PR[GP1:90,1] + -54.800;
   1:  PR[GP1:91,2] = PR[GP1:90,2] + 30.925;
   1:L PR[91] R[100]mm/sec CNT100;
   1:  PR[GP1:91,1] = PR[GP1:90,1] + -62.825;
   1:  PR[GP1:91,2] = PR[GP1:90,2] + 25.000;
   1:L PR[91] R[100]mm/sec CNT100;
   1:  PR[GP1:91,1] = PR[GP1:90,1] + -64.080;
   1:  PR[GP1:91,2] = PR[GP1:90,2] + 24.243;
   1:L PR[91] R[100]mm/sec CNT100;
   1:  PR[GP1:91,1] = PR[GP1:90,1] + -65.089;
   1:  PR[GP1:91,2] = PR[GP1:90,2] + 23.341;
   1:L PR[91] R[100]mm/sec CNT100;
   1:  PR[GP1:91,1] = PR[GP1:90,1] + -70.399;
   1:  PR[GP1:91,2] = PR[GP1:90,2] + 14.889;
   1:L PR[91] R[100]mm/sec CNT100;
   1:  PR[GP1:91,1] = PR[GP1:90,1] + -71.291;
   1:  PR[GP1:91,2] = PR[GP1:90,2] + 13.726;
   1:L PR[91] R[100]mm/sec CNT100;
   1:  PR[GP1:91,1] = PR[GP1:90,1] + -71.901;
   1:  PR[GP1:91,2] = PR[GP1:90,2] + 12.517;
   1:L PR[91] R[100]mm/sec CNT100;
   1:  PR[GP1:91,1] = PR[GP1:90,1] + -73.756;
   1:  PR[GP1:91,2] = PR[GP1:90,2] + 2.713;
   1:L PR[91] R[100]mm/sec CNT100;
   1:  PR[GP1:91,1] = PR[GP1:90,1] + -74.162;
   1:  PR[GP1:91,2] = PR[GP1:90,2] + 1.304;
   1:L PR[91] R[100]mm/sec CNT100;
   1:  PR[GP1:91,1] = PR[GP1:90,1] + -74.288;
   1:  PR[GP1:91,2] = PR[GP1:90,2] + -0.044;
   1:L PR[91] R[100]mm/sec CNT100;
   1:  PR[GP1:91,1] = PR[GP1:90,1] + -72.433;
   1:  PR[GP1:91,2] = PR[GP1:90,2] + -9.848;
   1:L PR[91] R[100]mm/sec CNT100;
   1:  PR[GP1:91,1] = PR[GP1:90,1] + -72.296;
   1:  PR[GP1:91,2] = PR[GP1:90,2] + -11.308;
   1:L PR[91] R[100]mm/sec CNT100;
   1:  PR[GP1:91,1] = PR[GP1:90,1] + -71.914;
   1:  PR[GP1:91,2] = PR[GP1:90,2] + -12.636;
   1:L PR[91] R[100]mm/sec CNT100;
   1:  PR[GP1:91,1] = PR[GP1:90,1] + -71.278;
   1:  PR[GP1:91,2] = PR[GP1:90,2] + -13.895;
   1:L PR[91] R[100]mm/sec CNT100;
   1:  PR[GP1:91,1] = PR[GP1:90,1] + -65.969;
   1:  PR[GP1:91,2] = PR[GP1:90,2] + -22.347;
   1:L PR[91] R[100]mm/sec CNT100;
   1:  PR[GP1:91,1] = PR[GP1:90,1] + -65.110;
   1:  PR[GP1:91,2] = PR[GP1:90,2] + -23.466;
   1:L PR[91] R[100]mm/sec CNT100;
   1:  PR[GP1:91,1] = PR[GP1:90,1] + -64.059;
   1:  PR[GP1:91,2] = PR[GP1:90,2] + -24.406;
   1:L PR[91] R[100]mm/sec CNT100;
   1:  PR[GP1:91,1] = PR[GP1:90,1] + -56.034;
   1:  PR[GP1:91,2] = PR[GP1:90,2] + -30.331;
   1:L PR[91] R[100]mm/sec CNT100;
   1:  PR[GP1:91,1] = PR[GP1:90,1] + -54.826;
   1:  PR[GP1:91,2] = PR[GP1:90,2] + -31.059;
   1:L PR[91] R[100]mm/sec CNT100;
   1:  PR[GP1:91,1] = PR[GP1:90,1] + -53.505;
   1:  PR[GP1:91,2] = PR[GP1:90,2] + -31.550;
   1:L PR[91] R[100]mm/sec CNT100;
   1:  PR[GP1:91,1] = PR[GP1:90,1] + -43.866;
   1:  PR[GP1:91,2] = PR[GP1:90,2] + -34.135;
   1:L PR[91] R[100]mm/sec CNT100;
   1:  PR[GP1:91,1] = PR[GP1:90,1] + -42.476;
   1:  PR[GP1:91,2] = PR[GP1:90,2] + -34.372;
   1:L PR[91] R[100]mm/sec CNT100;
   1:  PR[GP1:91,1] = PR[GP1:90,1] + -41.066;
   1:  PR[GP1:91,2] = PR[GP1:90,2] + -34.346;
   1:L PR[91] R[100]mm/sec CNT100;
   1:  PR[GP1:91,1] = PR[GP1:90,1] + -31.150;
   1:  PR[GP1:91,2] = PR[GP1:90,2] + -33.233;
   1:L PR[91] R[100]mm/sec CNT100;
   1:  PR[GP1:91,1] = PR[GP1:90,1] + -29.769;
   1:  PR[GP1:91,2] = PR[GP1:90,2] + -32.946;
   1:L PR[91] R[100]mm/sec CNT100;
   1:  PR[GP1:91,1] = PR[GP1:90,1] + -28.466;
   1:  PR[GP1:91,2] = PR[GP1:90,2] + -32.407;
   1:L PR[91] R[100]mm/sec CNT100;
   1:  PR[GP1:91,1] = PR[GP1:90,1] + -19.645;
   1:  PR[GP1:91,2] = PR[GP1:90,2] + -27.750;
   1:L PR[91] R[100]mm/sec CNT100;
   1:  PR[GP1:91,1] = PR[GP1:90,1] + -18.465;
   1:  PR[GP1:91,2] = PR[GP1:90,2] + -26.979;
   1:L PR[91] R[100]mm/sec CNT100;
   1:  PR[GP1:91,1] = PR[GP1:90,1] + -17.448;
   1:  PR[GP1:91,2] = PR[GP1:90,2] + -26.001;
   1:L PR[91] R[100]mm/sec CNT100;
   1:  PR[GP1:91,1] = PR[GP1:90,1] + -10.934;
   1:  PR[GP1:91,2] = PR[GP1:90,2] + -18.441;
   1:L PR[91] R[100]mm/sec CNT100;
   1:  PR[GP1:91,1] = PR[GP1:90,1] + -10.117;
   1:  PR[GP1:91,2] = PR[GP1:90,2] + -17.291;
   1:L PR[91] R[100]mm/sec CNT100;
   1:  PR[GP1:91,1] = PR[GP1:90,1] + -9.528;
   1:  PR[GP1:91,2] = PR[GP1:90,2] + -16.010;
   1:L PR[91] R[100]mm/sec CNT100;
   1:  PR[GP1:91,1] = PR[GP1:90,1] + -6.226;
   1:  PR[GP1:91,2] = PR[GP1:90,2] + -6.600;
   1:L PR[91] R[100]mm/sec CNT100;
   1:  PR[GP1:91,1] = PR[GP1:90,1] + -5.853;
   1:  PR[GP1:91,2] = PR[GP1:90,2] + -5.100;
   1:L PR[91] R[100]mm/sec CNT100;
   1:  PR[GP1:91,1] = PR[GP1:90,1] + -4.023;
   1:  PR[GP1:91,2] = PR[GP1:90,2] + -1.796;
   1:L PR[91] R[100]mm/sec CNT100;
   1:  PR[GP1:91,1] = PR[GP1:90,1] + -0.454;
   1:  PR[GP1:91,2] = PR[GP1:90,2] + -0.472;
   1:L PR[91] R[100]mm/sec CNT100;
   1:  PR[GP1:91,1] = PR[GP1:90,1] + 0.667;
   1:L PR[91] R[100]mm/sec CNT100;
   1:  PR[GP1:91,1] = PR[GP1:90,1] + 4.236;
   1:  PR[GP1:91,2] = PR[GP1:90,2] + -1.796;
   1:L PR[91] R[100]mm/sec CNT100;
   1:  PR[GP1:91,1] = PR[GP1:90,1] + 6.052;
   1:  PR[GP1:91,2] = PR[GP1:90,2] + -5.076;
   1:L PR[91] R[100]mm/sec CNT100;
   1:  PR[GP1:91,1] = PR[GP1:90,1] + 9.398;
   1:  PR[GP1:91,2] = PR[GP1:90,2] + -14.613;
   1:L PR[91] R[100]mm/sec CNT100;
   1:  PR[GP1:91,1] = PR[GP1:90,1] + 9.753;
   1:  PR[GP1:91,2] = PR[GP1:90,2] + -16.036;
   1:L PR[91] R[100]mm/sec CNT100;
   1:  PR[GP1:91,1] = PR[GP1:90,1] + 10.318;
   1:  PR[GP1:91,2] = PR[GP1:90,2] + -17.266;
   1:L PR[91] R[100]mm/sec CNT100;
   1:  PR[GP1:91,1] = PR[GP1:90,1] + 16.832;
   1:  PR[GP1:91,2] = PR[GP1:90,2] + -24.826;
   1:L PR[91] R[100]mm/sec CNT100;
   1:  PR[GP1:91,1] = PR[GP1:90,1] + 17.682;
   1:  PR[GP1:91,2] = PR[GP1:90,2] + -26.021;
   1:L PR[91] R[100]mm/sec CNT100;
   1:  PR[GP1:91,1] = PR[GP1:90,1] + 18.657;
   1:  PR[GP1:91,2] = PR[GP1:90,2] + -26.959;
   1:L PR[91] R[100]mm/sec CNT100;
   1:  PR[GP1:91,1] = PR[GP1:90,1] + 27.478;
   1:  PR[GP1:91,2] = PR[GP1:90,2] + -31.615;
   1:L PR[91] R[100]mm/sec CNT100;
   1:  PR[GP1:91,1] = PR[GP1:90,1] + 28.705;
   1:  PR[GP1:91,2] = PR[GP1:90,2] + -32.417;
   1:L PR[91] R[100]mm/sec CNT100;
   1:  PR[GP1:91,1] = PR[GP1:90,1] + 29.956;
   1:  PR[GP1:91,2] = PR[GP1:90,2] + -32.935;
   1:L PR[91] R[100]mm/sec CNT100;
   1:  PR[GP1:91,1] = PR[GP1:90,1] + 39.872;
   1:  PR[GP1:91,2] = PR[GP1:90,2] + -34.048;
   1:L PR[91] R[100]mm/sec CNT100;
   1:  PR[GP1:91,1] = PR[GP1:90,1] + 41.308;
   1:  PR[GP1:91,2] = PR[GP1:90,2] + -34.347;
   1:L PR[91] R[100]mm/sec CNT100;
   1:  PR[GP1:91,1] = PR[GP1:90,1] + 42.661;
   1:  PR[GP1:91,2] = PR[GP1:90,2] + -34.371;
   1:L PR[91] R[100]mm/sec CNT100;
   1:  PR[GP1:91,1] = PR[GP1:90,1] + 52.299;
   1:  PR[GP1:91,2] = PR[GP1:90,2] + -31.786;
   1:L PR[91] R[100]mm/sec CNT100;
   1:  PR[GP1:91,1] = PR[GP1:90,1] + 53.744;
   1:  PR[GP1:91,2] = PR[GP1:90,2] + -31.540;
   1:L PR[91] R[100]mm/sec CNT100;
   1:  PR[GP1:91,1] = PR[GP1:90,1] + 55.013;
   1:  PR[GP1:91,2] = PR[GP1:90,2] + -31.069;
   1:L PR[91] R[100]mm/sec CNT100;
   1:  PR[GP1:91,1] = PR[GP1:90,1] + 63.038;
   1:  PR[GP1:91,2] = PR[GP1:90,2] + -25.144;
   1:L PR[91] R[100]mm/sec CNT100;
   1:  PR[GP1:91,1] = PR[GP1:90,1] + 64.293;
   1:  PR[GP1:91,2] = PR[GP1:90,2] + -24.387;
   1:L PR[91] R[100]mm/sec CNT100;
   1:  PR[GP1:91,1] = PR[GP1:90,1] + 65.302;
   1:  PR[GP1:91,2] = PR[GP1:90,2] + -23.485;
   1:L PR[91] R[100]mm/sec CNT100;
   1:  PR[GP1:91,1] = PR[GP1:90,1] + 70.612;
   1:  PR[GP1:91,2] = PR[GP1:90,2] + -15.033;
   1:L PR[91] R[100]mm/sec CNT100;
   1:  PR[GP1:91,1] = PR[GP1:90,1] + 71.504;
   1:  PR[GP1:91,2] = PR[GP1:90,2] + -13.870;
   1:L PR[91] R[100]mm/sec CNT100;
   1:  PR[GP1:91,1] = PR[GP1:90,1] + 72.114;
   1:  PR[GP1:91,2] = PR[GP1:90,2] + -12.661;
   1:L PR[91] R[100]mm/sec CNT100;
   1:  PR[GP1:91,1] = PR[GP1:90,1] + 73.969;
   1:  PR[GP1:91,2] = PR[GP1:90,2] + -2.857;
   1:L PR[91] R[100]mm/sec CNT100;
   1:  PR[GP1:91,1] = PR[GP1:90,1] + 74.375;
   1:  PR[GP1:91,2] = PR[GP1:90,2] + -1.448;
   1:L PR[91] R[100]mm/sec CNT100;
   1:  PR[GP1:91,1] = PR[GP1:90,1] + 74.501;
   1:  PR[GP1:91,2] = PR[GP1:90,2] + -0.100;
   1:L PR[91] R[100]mm/sec CNT100;
   1:  PR[GP1:91,1] = PR[GP1:90,1] + 72.646;
   1:  PR[GP1:91,2] = PR[GP1:90,2] + 9.704;
   1:L PR[91] R[100]mm/sec CNT100;
   1:  PR[GP1:91,1] = PR[GP1:90,1] + 72.509;
   1:  PR[GP1:91,2] = PR[GP1:90,2] + 11.164;
   1:L PR[91] R[100]mm/sec CNT100;
   1:  PR[GP1:91,1] = PR[GP1:90,1] + 72.127;
   1:  PR[GP1:91,2] = PR[GP1:90,2] + 12.492;
   1:L PR[91] R[100]mm/sec CNT100;
   1:  PR[GP1:91,1] = PR[GP1:90,1] + 71.492;
   1:  PR[GP1:91,2] = PR[GP1:90,2] + 13.751;
   1:L PR[91] R[100]mm/sec CNT100;
   1:  PR[GP1:91,1] = PR[GP1:90,1] + 66.182;
   1:  PR[GP1:91,2] = PR[GP1:90,2] + 22.203;
   1:L PR[91] R[100]mm/sec CNT100;
   1:  PR[GP1:91,1] = PR[GP1:90,1] + 65.324;
   1:  PR[GP1:91,2] = PR[GP1:90,2] + 23.322;
   1:L PR[91] R[100]mm/sec CNT100;
   1:  PR[GP1:91,1] = PR[GP1:90,1] + 64.272;
   1:  PR[GP1:91,2] = PR[GP1:90,2] + 24.262;
   1:L PR[91] R[100]mm/sec CNT100;
   1:  PR[GP1:91,1] = PR[GP1:90,1] + 56.247;
   1:  PR[GP1:91,2] = PR[GP1:90,2] + 30.186;
   1:L PR[91] R[100]mm/sec CNT100;
   1:  PR[GP1:91,1] = PR[GP1:90,1] + 55.040;
   1:  PR[GP1:91,2] = PR[GP1:90,2] + 30.915;
   1:L PR[91] R[100]mm/sec CNT100;
   1:  PR[GP1:91,1] = PR[GP1:90,1] + 53.718;
   1:  PR[GP1:91,2] = PR[GP1:90,2] + 31.406;
   1:L PR[91] R[100]mm/sec CNT100;
   1:  PR[GP1:91,1] = PR[GP1:90,1] + 44.079;
   1:  PR[GP1:91,2] = PR[GP1:90,2] + 33.991;
   1:L PR[91] R[100]mm/sec CNT100;
   1:  PR[GP1:91,1] = PR[GP1:90,1] + 42.689;
   1:  PR[GP1:91,2] = PR[GP1:90,2] + 34.228;
   1:L PR[91] R[100]mm/sec CNT100;
   1:  PR[GP1:91,1] = PR[GP1:90,1] + 41.279;
   1:  PR[GP1:91,2] = PR[GP1:90,2] + 34.202;
   1:L PR[91] R[100]mm/sec CNT100;
   1:  PR[GP1:91,1] = PR[GP1:90,1] + 31.363;
   1:  PR[GP1:91,2] = PR[GP1:90,2] + 33.089;
   1:L PR[91] R[100]mm/sec CNT100;
   1:  PR[GP1:91,1] = PR[GP1:90,1] + 29.982;
   1:  PR[GP1:91,2] = PR[GP1:90,2] + 32.802;
   1:L PR[91] R[100]mm/sec CNT100;
   1:  PR[GP1:91,1] = PR[GP1:90,1] + 28.679;
   1:  PR[GP1:91,2] = PR[GP1:90,2] + 32.263;
   1:L PR[91] R[100]mm/sec CNT100;
   1:  PR[GP1:91,1] = PR[GP1:90,1] + 19.858;
   1:  PR[GP1:91,2] = PR[GP1:90,2] + 27.606;
   1:L PR[91] R[100]mm/sec CNT100;
   1:  PR[GP1:91,1] = PR[GP1:90,1] + 18.678;
   1:  PR[GP1:91,2] = PR[GP1:90,2] + 26.835;
   1:L PR[91] R[100]mm/sec CNT100;
   1:  PR[GP1:91,1] = PR[GP1:90,1] + 17.662;
   1:  PR[GP1:91,2] = PR[GP1:90,2] + 25.857;
   1:L PR[91] R[100]mm/sec CNT100;
   1:  PR[GP1:91,1] = PR[GP1:90,1] + 11.147;
   1:  PR[GP1:91,2] = PR[GP1:90,2] + 18.297;
   1:L PR[91] R[100]mm/sec CNT100;
   1:  PR[GP1:91,1] = PR[GP1:90,1] + 10.330;
   1:  PR[GP1:91,2] = PR[GP1:90,2] + 17.147;
   1:L PR[91] R[100]mm/sec CNT100;
   1:  PR[GP1:91,1] = PR[GP1:90,1] + 9.741;
   1:  PR[GP1:91,2] = PR[GP1:90,2] + 15.866;
   1:L PR[91] R[100]mm/sec CNT100;
   1:  PR[GP1:91,1] = PR[GP1:90,1] + 6.439;
   1:  PR[GP1:91,2] = PR[GP1:90,2] + 6.456;
   1:L PR[91] R[100]mm/sec CNT100;
   1:  PR[GP1:91,1] = PR[GP1:90,1] + 6.066;
   1:  PR[GP1:91,2] = PR[GP1:90,2] + 4.956;
   1:L PR[91] R[100]mm/sec CNT100;
   1:  PR[GP1:91,1] = PR[GP1:90,1] + 4.236;
   1:  PR[GP1:91,2] = PR[GP1:90,2] + 1.652;
   1:L PR[91] R[100]mm/sec CNT100;
   1:  PR[GP1:91,1] = PR[GP1:90,1] + 0.667;
   1:  PR[GP1:91,2] = PR[GP1:90,2] + 0.328;
   1:L PR[91] R[100]mm/sec CNT100;
   1:  PR[GP1:91,1] = PR[GP1:90,1] + -0.454;
   1:L PR[91] R[100]mm/sec CNT100;
   1:  ! -- Layer/Ebene 4 -- !;
   1:  PR[91] = PR[90];
   1:  PR[GP1:91,1] = PR[GP1:90,1] + -4.023;
   1:  PR[GP1:91,2] = PR[GP1:90,2] + 1.652;
   1:  PR[GP1:91,3] = PR[GP1:90,3] + 2.745;
   1:L PR[91] R[100]mm/sec CNT100;
   1:  PR[GP1:91,1] = PR[GP1:90,1] + -5.839;
   1:  PR[GP1:91,2] = PR[GP1:90,2] + 4.932;
   1:L PR[91] R[100]mm/sec CNT100;
   1:  PR[GP1:91,1] = PR[GP1:90,1] + -8.857;
   1:  PR[GP1:91,2] = PR[GP1:90,2] + 13.533;
   1:L PR[91] R[100]mm/sec CNT100;
   1:  PR[GP1:91,1] = PR[GP1:90,1] + -9.332;
   1:  PR[GP1:91,2] = PR[GP1:90,2] + 15.440;
   1:L PR[91] R[100]mm/sec CNT100;
   1:  PR[GP1:91,1] = PR[GP1:90,1] + -10.105;
   1:  PR[GP1:91,2] = PR[GP1:90,2] + 17.122;
   1:L PR[91] R[100]mm/sec CNT100;
   1:  PR[GP1:91,1] = PR[GP1:90,1] + -15.972;
   1:  PR[GP1:91,2] = PR[GP1:90,2] + 23.930;
   1:L PR[91] R[100]mm/sec CNT100;
   1:  PR[GP1:91,1] = PR[GP1:90,1] + -17.110;
   1:  PR[GP1:91,2] = PR[GP1:90,2] + 25.532;
   1:L PR[91] R[100]mm/sec CNT100;
   1:  PR[GP1:91,1] = PR[GP1:90,1] + -18.444;
   1:  PR[GP1:91,2] = PR[GP1:90,2] + 26.815;
   1:L PR[91] R[100]mm/sec CNT100;
   1:  PR[GP1:91,1] = PR[GP1:90,1] + -26.388;
   1:  PR[GP1:91,2] = PR[GP1:90,2] + 31.008;
   1:L PR[91] R[100]mm/sec CNT100;
   1:  PR[GP1:91,1] = PR[GP1:90,1] + -28.032;
   1:  PR[GP1:91,2] = PR[GP1:90,2] + 32.083;
   1:L PR[91] R[100]mm/sec CNT100;
   1:  PR[GP1:91,1] = PR[GP1:90,1] + -29.743;
   1:  PR[GP1:91,2] = PR[GP1:90,2] + 32.791;
   1:L PR[91] R[100]mm/sec CNT100;
   1:  PR[GP1:91,1] = PR[GP1:90,1] + -38.673;
   1:  PR[GP1:91,2] = PR[GP1:90,2] + 33.794;
   1:L PR[91] R[100]mm/sec CNT100;
   1:  PR[GP1:91,1] = PR[GP1:90,1] + -40.597;
   1:  PR[GP1:91,2] = PR[GP1:90,2] + 34.194;
   1:L PR[91] R[100]mm/sec CNT100;
   1:  PR[GP1:91,1] = PR[GP1:90,1] + -42.448;
   1:  PR[GP1:91,2] = PR[GP1:90,2] + 34.227;
   1:L PR[91] R[100]mm/sec CNT100;
   1:  PR[GP1:91,1] = PR[GP1:90,1] + -51.128;
   1:  PR[GP1:91,2] = PR[GP1:90,2] + 31.899;
   1:L PR[91] R[100]mm/sec CNT100;
   1:  PR[GP1:91,1] = PR[GP1:90,1] + -53.064;
   1:  PR[GP1:91,2] = PR[GP1:90,2] + 31.569;
   1:L PR[91] R[100]mm/sec CNT100;
   1:  PR[GP1:91,1] = PR[GP1:90,1] + -54.800;
   1:  PR[GP1:91,2] = PR[GP1:90,2] + 30.925;
   1:L PR[91] R[100]mm/sec CNT100;
   1:  PR[GP1:91,1] = PR[GP1:90,1] + -62.027;
   1:  PR[GP1:91,2] = PR[GP1:90,2] + 25.589;
   1:L PR[91] R[100]mm/sec CNT100;
   1:  PR[GP1:91,1] = PR[GP1:90,1] + -63.709;
   1:  PR[GP1:91,2] = PR[GP1:90,2] + 24.575;
   1:L PR[91] R[100]mm/sec CNT100;
   1:  PR[GP1:91,1] = PR[GP1:90,1] + -65.090;
   1:  PR[GP1:91,2] = PR[GP1:90,2] + 23.340;
   1:L PR[91] R[100]mm/sec CNT100;
   1:  PR[GP1:91,1] = PR[GP1:90,1] + -69.871;
   1:  PR[GP1:91,2] = PR[GP1:90,2] + 15.729;
   1:L PR[91] R[100]mm/sec CNT100;
   1:  PR[GP1:91,1] = PR[GP1:90,1] + -71.067;
   1:  PR[GP1:91,2] = PR[GP1:90,2] + 14.170;
   1:L PR[91] R[100]mm/sec CNT100;
   1:  PR[GP1:91,1] = PR[GP1:90,1] + -71.901;
   1:  PR[GP1:91,2] = PR[GP1:90,2] + 12.517;
   1:L PR[91] R[100]mm/sec CNT100;
   1:  PR[GP1:91,1] = PR[GP1:90,1] + -73.572;
   1:  PR[GP1:91,2] = PR[GP1:90,2] + 3.688;
   1:L PR[91] R[100]mm/sec CNT100;
   1:  PR[GP1:91,1] = PR[GP1:90,1] + -74.115;
   1:  PR[GP1:91,2] = PR[GP1:90,2] + 1.800;
   1:L PR[91] R[100]mm/sec CNT100;
   1:  PR[GP1:91,1] = PR[GP1:90,1] + -74.288;
   1:  PR[GP1:91,2] = PR[GP1:90,2] + -0.044;
   1:L PR[91] R[100]mm/sec CNT100;
   1:  PR[GP1:91,1] = PR[GP1:90,1] + -72.617;
   1:  PR[GP1:91,2] = PR[GP1:90,2] + -8.873;
   1:L PR[91] R[100]mm/sec CNT100;
   1:  PR[GP1:91,1] = PR[GP1:90,1] + -72.434;
   1:  PR[GP1:91,2] = PR[GP1:90,2] + -10.829;
   1:L PR[91] R[100]mm/sec CNT100;
   1:  PR[GP1:91,1] = PR[GP1:90,1] + -71.914;
   1:  PR[GP1:91,2] = PR[GP1:90,2] + -12.636;
   1:L PR[91] R[100]mm/sec CNT100;
   1:  PR[GP1:91,1] = PR[GP1:90,1] + -71.054;
   1:  PR[GP1:91,2] = PR[GP1:90,2] + -14.339;
   1:L PR[91] R[100]mm/sec CNT100;
   1:  PR[GP1:91,1] = PR[GP1:90,1] + -66.272;
   1:  PR[GP1:91,2] = PR[GP1:90,2] + -21.951;
   1:L PR[91] R[100]mm/sec CNT100;
   1:  PR[GP1:91,1] = PR[GP1:90,1] + -65.111;
   1:  PR[GP1:91,2] = PR[GP1:90,2] + -23.465;
   1:L PR[91] R[100]mm/sec CNT100;
   1:  PR[GP1:91,1] = PR[GP1:90,1] + -63.688;
   1:  PR[GP1:91,2] = PR[GP1:90,2] + -24.737;
   1:L PR[91] R[100]mm/sec CNT100;
   1:  PR[GP1:91,1] = PR[GP1:90,1] + -56.461;
   1:  PR[GP1:91,2] = PR[GP1:90,2] + -30.073;
   1:L PR[91] R[100]mm/sec CNT100;
   1:  PR[GP1:91,1] = PR[GP1:90,1] + -54.827;
   1:  PR[GP1:91,2] = PR[GP1:90,2] + -31.059;
   1:L PR[91] R[100]mm/sec CNT100;
   1:  PR[GP1:91,1] = PR[GP1:90,1] + -53.038;
   1:  PR[GP1:91,2] = PR[GP1:90,2] + -31.723;
   1:L PR[91] R[100]mm/sec CNT100;
   1:  PR[GP1:91,1] = PR[GP1:90,1] + -44.358;
   1:  PR[GP1:91,2] = PR[GP1:90,2] + -34.051;
   1:L PR[91] R[100]mm/sec CNT100;
   1:  PR[GP1:91,1] = PR[GP1:90,1] + -42.476;
   1:  PR[GP1:91,2] = PR[GP1:90,2] + -34.372;
   1:L PR[91] R[100]mm/sec CNT100;
   1:  PR[GP1:91,1] = PR[GP1:90,1] + -40.568;
   1:  PR[GP1:91,2] = PR[GP1:90,2] + -34.337;
   1:L PR[91] R[100]mm/sec CNT100;
   1:  PR[GP1:91,1] = PR[GP1:90,1] + -31.638;
   1:  PR[GP1:91,2] = PR[GP1:90,2] + -33.334;
   1:L PR[91] R[100]mm/sec CNT100;
   1:  PR[GP1:91,1] = PR[GP1:90,1] + -29.769;
   1:  PR[GP1:91,2] = PR[GP1:90,2] + -32.946;
   1:L PR[91] R[100]mm/sec CNT100;
   1:  PR[GP1:91,1] = PR[GP1:90,1] + -28.006;
   1:  PR[GP1:91,2] = PR[GP1:90,2] + -32.217;
   1:L PR[91] R[100]mm/sec CNT100;
   1:  PR[GP1:91,1] = PR[GP1:90,1] + -20.062;
   1:  PR[GP1:91,2] = PR[GP1:90,2] + -28.023;
   1:L PR[91] R[100]mm/sec CNT100;
   1:  PR[GP1:91,1] = PR[GP1:90,1] + -18.465;
   1:  PR[GP1:91,2] = PR[GP1:90,2] + -26.979;
   1:L PR[91] R[100]mm/sec CNT100;
   1:  PR[GP1:91,1] = PR[GP1:90,1] + -17.089;
   1:  PR[GP1:91,2] = PR[GP1:90,2] + -25.656;
   1:L PR[91] R[100]mm/sec CNT100;
   1:  PR[GP1:91,1] = PR[GP1:90,1] + -11.223;
   1:  PR[GP1:91,2] = PR[GP1:90,2] + -18.847;
   1:L PR[91] R[100]mm/sec CNT100;
   1:  PR[GP1:91,1] = PR[GP1:90,1] + -10.117;
   1:  PR[GP1:91,2] = PR[GP1:90,2] + -17.292;
   1:L PR[91] R[100]mm/sec CNT100;
   1:  PR[GP1:91,1] = PR[GP1:90,1] + -9.320;
   1:  PR[GP1:91,2] = PR[GP1:90,2] + -15.558;
   1:L PR[91] R[100]mm/sec CNT100;
   1:  PR[GP1:91,1] = PR[GP1:90,1] + -6.346;
   1:  PR[GP1:91,2] = PR[GP1:90,2] + -7.083;
   1:L PR[91] R[100]mm/sec CNT100;
   1:  PR[GP1:91,1] = PR[GP1:90,1] + -5.853;
   1:  PR[GP1:91,2] = PR[GP1:90,2] + -5.100;
   1:L PR[91] R[100]mm/sec CNT100;
   1:  PR[GP1:91,1] = PR[GP1:90,1] + -4.023;
   1:  PR[GP1:91,2] = PR[GP1:90,2] + -1.796;
   1:L PR[91] R[100]mm/sec CNT100;
   1:  PR[GP1:91,1] = PR[GP1:90,1] + -0.454;
   1:  PR[GP1:91,2] = PR[GP1:90,2] + -0.472;
   1:L PR[91] R[100]mm/sec CNT100;
   1:  PR[GP1:91,1] = PR[GP1:90,1] + 0.667;
   1:L PR[91] R[100]mm/sec CNT100;
   1:  PR[GP1:91,1] = PR[GP1:90,1] + 4.236;
   1:  PR[GP1:91,2] = PR[GP1:90,2] + -1.796;
   1:L PR[91] R[100]mm/sec CNT100;
   1:  PR[GP1:91,1] = PR[GP1:90,1] + 6.052;
   1:  PR[GP1:91,2] = PR[GP1:90,2] + -5.076;
   1:L PR[91] R[100]mm/sec CNT100;
   1:  PR[GP1:91,1] = PR[GP1:90,1] + 9.070;
   1:  PR[GP1:91,2] = PR[GP1:90,2] + -13.677;
   1:L PR[91] R[100]mm/sec CNT100;
   1:  PR[GP1:91,1] = PR[GP1:90,1] + 9.545;
   1:  PR[GP1:91,2] = PR[GP1:90,2] + -15.584;
   1:L PR[91] R[100]mm/sec CNT100;
   1:  PR[GP1:91,1] = PR[GP1:90,1] + 10.318;
   1:  PR[GP1:91,2] = PR[GP1:90,2] + -17.266;
   1:L PR[91] R[100]mm/sec CNT100;
   1:  PR[GP1:91,1] = PR[GP1:90,1] + 16.185;
   1:  PR[GP1:91,2] = PR[GP1:90,2] + -24.074;
   1:L PR[91] R[100]mm/sec CNT100;
   1:  PR[GP1:91,1] = PR[GP1:90,1] + 17.323;
   1:  PR[GP1:91,2] = PR[GP1:90,2] + -25.676;
   1:L PR[91] R[100]mm/sec CNT100;
   1:  PR[GP1:91,1] = PR[GP1:90,1] + 18.658;
   1:  PR[GP1:91,2] = PR[GP1:90,2] + -26.959;
   1:L PR[91] R[100]mm/sec CNT100;
   1:  PR[GP1:91,1] = PR[GP1:90,1] + 26.601;
   1:  PR[GP1:91,2] = PR[GP1:90,2] + -31.152;
   1:L PR[91] R[100]mm/sec CNT100;
   1:  PR[GP1:91,1] = PR[GP1:90,1] + 28.245;
   1:  PR[GP1:91,2] = PR[GP1:90,2] + -32.227;
   1:L PR[91] R[100]mm/sec CNT100;
   1:  PR[GP1:91,1] = PR[GP1:90,1] + 29.957;
   1:  PR[GP1:91,2] = PR[GP1:90,2] + -32.935;
   1:L PR[91] R[100]mm/sec CNT100;
   1:  PR[GP1:91,1] = PR[GP1:90,1] + 38.887;
   1:  PR[GP1:91,2] = PR[GP1:90,2] + -33.938;
   1:L PR[91] R[100]mm/sec CNT100;
   1:  PR[GP1:91,1] = PR[GP1:90,1] + 40.810;
   1:  PR[GP1:91,2] = PR[GP1:90,2] + -34.338;
   1:L PR[91] R[100]mm/sec CNT100;
   1:  PR[GP1:91,1] = PR[GP1:90,1] + 42.661;
   1:  PR[GP1:91,2] = PR[GP1:90,2] + -34.371;
   1:L PR[91] R[100]mm/sec CNT100;
   1:  PR[GP1:91,1] = PR[GP1:90,1] + 51.341;
   1:  PR[GP1:91,2] = PR[GP1:90,2] + -32.043;
   1:L PR[91] R[100]mm/sec CNT100;
   1:  PR[GP1:91,1] = PR[GP1:90,1] + 53.278;
   1:  PR[GP1:91,2] = PR[GP1:90,2] + -31.713;
   1:L PR[91] R[100]mm/sec CNT100;
   1:  PR[GP1:91,1] = PR[GP1:90,1] + 55.013;
   1:  PR[GP1:91,2] = PR[GP1:90,2] + -31.069;
   1:L PR[91] R[100]mm/sec CNT100;
   1:  PR[GP1:91,1] = PR[GP1:90,1] + 62.240;
   1:  PR[GP1:91,2] = PR[GP1:90,2] + -25.733;
   1:L PR[91] R[100]mm/sec CNT100;
   1:  PR[GP1:91,1] = PR[GP1:90,1] + 63.922;
   1:  PR[GP1:91,2] = PR[GP1:90,2] + -24.719;
   1:L PR[91] R[100]mm/sec CNT100;
   1:  PR[GP1:91,1] = PR[GP1:90,1] + 65.303;
   1:  PR[GP1:91,2] = PR[GP1:90,2] + -23.484;
   1:L PR[91] R[100]mm/sec CNT100;
   1:  PR[GP1:91,1] = PR[GP1:90,1] + 70.084;
   1:  PR[GP1:91,2] = PR[GP1:90,2] + -15.873;
   1:L PR[91] R[100]mm/sec CNT100;
   1:  PR[GP1:91,1] = PR[GP1:90,1] + 71.280;
   1:  PR[GP1:91,2] = PR[GP1:90,2] + -14.314;
   1:L PR[91] R[100]mm/sec CNT100;
   1:  PR[GP1:91,1] = PR[GP1:90,1] + 72.114;
   1:  PR[GP1:91,2] = PR[GP1:90,2] + -12.661;
   1:L PR[91] R[100]mm/sec CNT100;
   1:  PR[GP1:91,1] = PR[GP1:90,1] + 73.785;
   1:  PR[GP1:91,2] = PR[GP1:90,2] + -3.832;
   1:L PR[91] R[100]mm/sec CNT100;
   1:  PR[GP1:91,1] = PR[GP1:90,1] + 74.329;
   1:  PR[GP1:91,2] = PR[GP1:90,2] + -1.944;
   1:L PR[91] R[100]mm/sec CNT100;
   1:  PR[GP1:91,1] = PR[GP1:90,1] + 74.501;
   1:  PR[GP1:91,2] = PR[GP1:90,2] + -0.100;
   1:L PR[91] R[100]mm/sec CNT100;
   1:  PR[GP1:91,1] = PR[GP1:90,1] + 72.831;
   1:  PR[GP1:91,2] = PR[GP1:90,2] + 8.729;
   1:L PR[91] R[100]mm/sec CNT100;
   1:  PR[GP1:91,1] = PR[GP1:90,1] + 72.647;
   1:  PR[GP1:91,2] = PR[GP1:90,2] + 10.685;
   1:L PR[91] R[100]mm/sec CNT100;
   1:  PR[GP1:91,1] = PR[GP1:90,1] + 72.127;
   1:  PR[GP1:91,2] = PR[GP1:90,2] + 12.492;
   1:L PR[91] R[100]mm/sec CNT100;
   1:  PR[GP1:91,1] = PR[GP1:90,1] + 71.267;
   1:  PR[GP1:91,2] = PR[GP1:90,2] + 14.195;
   1:L PR[91] R[100]mm/sec CNT100;
   1:  PR[GP1:91,1] = PR[GP1:90,1] + 66.485;
   1:  PR[GP1:91,2] = PR[GP1:90,2] + 21.807;
   1:L PR[91] R[100]mm/sec CNT100;
   1:  PR[GP1:91,1] = PR[GP1:90,1] + 65.324;
   1:  PR[GP1:91,2] = PR[GP1:90,2] + 23.321;
   1:L PR[91] R[100]mm/sec CNT100;
   1:  PR[GP1:91,1] = PR[GP1:90,1] + 63.901;
   1:  PR[GP1:91,2] = PR[GP1:90,2] + 24.593;
   1:L PR[91] R[100]mm/sec CNT100;
   1:  PR[GP1:91,1] = PR[GP1:90,1] + 56.674;
   1:  PR[GP1:91,2] = PR[GP1:90,2] + 29.929;
   1:L PR[91] R[100]mm/sec CNT100;
   1:  PR[GP1:91,1] = PR[GP1:90,1] + 55.040;
   1:  PR[GP1:91,2] = PR[GP1:90,2] + 30.915;
   1:L PR[91] R[100]mm/sec CNT100;
   1:  PR[GP1:91,1] = PR[GP1:90,1] + 53.251;
   1:  PR[GP1:91,2] = PR[GP1:90,2] + 31.579;
   1:L PR[91] R[100]mm/sec CNT100;
   1:  PR[GP1:91,1] = PR[GP1:90,1] + 44.571;
   1:  PR[GP1:91,2] = PR[GP1:90,2] + 33.907;
   1:L PR[91] R[100]mm/sec CNT100;
   1:  PR[GP1:91,1] = PR[GP1:90,1] + 42.690;
   1:  PR[GP1:91,2] = PR[GP1:90,2] + 34.228;
   1:L PR[91] R[100]mm/sec CNT100;
   1:  PR[GP1:91,1] = PR[GP1:90,1] + 40.782;
   1:  PR[GP1:91,2] = PR[GP1:90,2] + 34.193;
   1:L PR[91] R[100]mm/sec CNT100;
   1:  PR[GP1:91,1] = PR[GP1:90,1] + 31.851;
   1:  PR[GP1:91,2] = PR[GP1:90,2] + 33.190;
   1:L PR[91] R[100]mm/sec CNT100;
   1:  PR[GP1:91,1] = PR[GP1:90,1] + 29.983;
   1:  PR[GP1:91,2] = PR[GP1:90,2] + 32.802;
   1:L PR[91] R[100]mm/sec CNT100;
   1:  PR[GP1:91,1] = PR[GP1:90,1] + 28.219;
   1:  PR[GP1:91,2] = PR[GP1:90,2] + 32.073;
   1:L PR[91] R[100]mm/sec CNT100;
   1:  PR[GP1:91,1] = PR[GP1:90,1] + 20.275;
   1:  PR[GP1:91,2] = PR[GP1:90,2] + 27.879;
   1:L PR[91] R[100]mm/sec CNT100;
   1:  PR[GP1:91,1] = PR[GP1:90,1] + 18.678;
   1:  PR[GP1:91,2] = PR[GP1:90,2] + 26.835;
   1:L PR[91] R[100]mm/sec CNT100;
   1:  PR[GP1:91,1] = PR[GP1:90,1] + 17.303;
   1:  PR[GP1:91,2] = PR[GP1:90,2] + 25.512;
   1:L PR[91] R[100]mm/sec CNT100;
   1:  PR[GP1:91,1] = PR[GP1:90,1] + 11.436;
   1:  PR[GP1:91,2] = PR[GP1:90,2] + 18.703;
   1:L PR[91] R[100]mm/sec CNT100;
   1:  PR[GP1:91,1] = PR[GP1:90,1] + 10.330;
   1:  PR[GP1:91,2] = PR[GP1:90,2] + 17.148;
   1:L PR[91] R[100]mm/sec CNT100;
   1:  PR[GP1:91,1] = PR[GP1:90,1] + 9.533;
   1:  PR[GP1:91,2] = PR[GP1:90,2] + 15.414;
   1:L PR[91] R[100]mm/sec CNT100;
   1:  PR[GP1:91,1] = PR[GP1:90,1] + 6.560;
   1:  PR[GP1:91,2] = PR[GP1:90,2] + 6.939;
   1:L PR[91] R[100]mm/sec CNT100;
   1:  PR[GP1:91,1] = PR[GP1:90,1] + 6.066;
   1:  PR[GP1:91,2] = PR[GP1:90,2] + 4.956;
   1:L PR[91] R[100]mm/sec CNT100;
   1:  PR[GP1:91,1] = PR[GP1:90,1] + 4.236;
   1:  PR[GP1:91,2] = PR[GP1:90,2] + 1.652;
   1:L PR[91] R[100]mm/sec CNT100;
   1:  PR[GP1:91,1] = PR[GP1:90,1] + 0.667;
   1:  PR[GP1:91,2] = PR[GP1:90,2] + 0.328;
   1:L PR[91] R[100]mm/sec CNT100;
   1:  PR[GP1:91,1] = PR[GP1:90,1] + -0.454;
   1:L PR[91] R[100]mm/sec CNT100;
   1:  ! -- Layer/Ebene 5 -- !;
   1:  PR[91] = PR[90];
   1:  PR[GP1:91,1] = PR[GP1:90,1] + -4.023;
   1:  PR[GP1:91,2] = PR[GP1:90,2] + 1.652;
   1:  PR[GP1:91,3] = PR[GP1:90,3] + 3.355;
   1:L PR[91] R[100]mm/sec CNT100;
   1:  PR[GP1:91,1] = PR[GP1:90,1] + -5.839;
   1:  PR[GP1:91,2] = PR[GP1:90,2] + 4.932;
   1:L PR[91] R[100]mm/sec CNT100;
   1:  PR[GP1:91,1] = PR[GP1:90,1] + -8.529;
   1:  PR[GP1:91,2] = PR[GP1:90,2] + 12.598;
   1:L PR[91] R[100]mm/sec CNT100;
   1:  PR[GP1:91,1] = PR[GP1:90,1] + -9.124;
   1:  PR[GP1:91,2] = PR[GP1:90,2] + 14.987;
   1:L PR[91] R[100]mm/sec CNT100;
   1:  PR[GP1:91,1] = PR[GP1:90,1] + -10.105;
   1:  PR[GP1:91,2] = PR[GP1:90,2] + 17.123;
   1:L PR[91] R[100]mm/sec CNT100;
   1:  PR[GP1:91,1] = PR[GP1:90,1] + -15.324;
   1:  PR[GP1:91,2] = PR[GP1:90,2] + 23.179;
   1:L PR[91] R[100]mm/sec CNT100;
   1:  PR[GP1:91,1] = PR[GP1:90,1] + -16.751;
   1:  PR[GP1:91,2] = PR[GP1:90,2] + 25.186;
   1:L PR[91] R[100]mm/sec CNT100;
   1:  PR[GP1:91,1] = PR[GP1:90,1] + -18.445;
   1:  PR[GP1:91,2] = PR[GP1:90,2] + 26.815;
   1:L PR[91] R[100]mm/sec CNT100;
   1:  PR[GP1:91,1] = PR[GP1:90,1] + -25.511;
   1:  PR[GP1:91,2] = PR[GP1:90,2] + 30.546;
   1:L PR[91] R[100]mm/sec CNT100;
   1:  PR[GP1:91,1] = PR[GP1:90,1] + -27.572;
   1:  PR[GP1:91,2] = PR[GP1:90,2] + 31.893;
   1:L PR[91] R[100]mm/sec CNT100;
   1:  PR[GP1:91,1] = PR[GP1:90,1] + -29.744;
   1:  PR[GP1:91,2] = PR[GP1:90,2] + 32.791;
   1:L PR[91] R[100]mm/sec CNT100;
   1:  PR[GP1:91,1] = PR[GP1:90,1] + -37.688;
   1:  PR[GP1:91,2] = PR[GP1:90,2] + 33.683;
   1:L PR[91] R[100]mm/sec CNT100;
   1:  PR[GP1:91,1] = PR[GP1:90,1] + -40.099;
   1:  PR[GP1:91,2] = PR[GP1:90,2] + 34.185;
   1:L PR[91] R[100]mm/sec CNT100;
   1:  PR[GP1:91,1] = PR[GP1:90,1] + -42.448;
   1:  PR[GP1:91,2] = PR[GP1:90,2] + 34.227;
   1:L PR[91] R[100]mm/sec CNT100;
   1:  PR[GP1:91,1] = PR[GP1:90,1] + -50.170;
   1:  PR[GP1:91,2] = PR[GP1:90,2] + 32.156;
   1:L PR[91] R[100]mm/sec CNT100;
   1:  PR[GP1:91,1] = PR[GP1:90,1] + -52.598;
   1:  PR[GP1:91,2] = PR[GP1:90,2] + 31.743;
   1:L PR[91] R[100]mm/sec CNT100;
   1:  PR[GP1:91,1] = PR[GP1:90,1] + -54.800;
   1:  PR[GP1:91,2] = PR[GP1:90,2] + 30.924;
   1:L PR[91] R[100]mm/sec CNT100;
   1:  PR[GP1:91,1] = PR[GP1:90,1] + -61.229;
   1:  PR[GP1:91,2] = PR[GP1:90,2] + 26.178;
   1:L PR[91] R[100]mm/sec CNT100;
   1:  PR[GP1:91,1] = PR[GP1:90,1] + -63.338;
   1:  PR[GP1:91,2] = PR[GP1:90,2] + 24.906;
   1:L PR[91] R[100]mm/sec CNT100;
   1:  PR[GP1:91,1] = PR[GP1:90,1] + -65.090;
   1:  PR[GP1:91,2] = PR[GP1:90,2] + 23.340;
   1:L PR[91] R[100]mm/sec CNT100;
   1:  PR[GP1:91,1] = PR[GP1:90,1] + -69.344;
   1:  PR[GP1:91,2] = PR[GP1:90,2] + 16.569;
   1:L PR[91] R[100]mm/sec CNT100;
   1:  PR[GP1:91,1] = PR[GP1:90,1] + -70.842;
   1:  PR[GP1:91,2] = PR[GP1:90,2] + 14.615;
   1:L PR[91] R[100]mm/sec CNT100;
   1:  PR[GP1:91,1] = PR[GP1:90,1] + -71.901;
   1:  PR[GP1:91,2] = PR[GP1:90,2] + 12.517;
   1:L PR[91] R[100]mm/sec CNT100;
   1:  PR[GP1:91,1] = PR[GP1:90,1] + -73.387;
   1:  PR[GP1:91,2] = PR[GP1:90,2] + 4.662;
   1:L PR[91] R[100]mm/sec CNT100;
   1:  PR[GP1:91,1] = PR[GP1:90,1] + -74.069;
   1:  PR[GP1:91,2] = PR[GP1:90,2] + 2.296;
   1:L PR[91] R[100]mm/sec CNT100;
   1:  PR[GP1:91,1] = PR[GP1:90,1] + -74.288;
   1:  PR[GP1:91,2] = PR[GP1:90,2] + -0.044;
   1:L PR[91] R[100]mm/sec CNT100;
   1:  PR[GP1:91,1] = PR[GP1:90,1] + -72.802;
   1:  PR[GP1:91,2] = PR[GP1:90,2] + -7.898;
   1:L PR[91] R[100]mm/sec CNT100;
   1:  PR[GP1:91,1] = PR[GP1:90,1] + -72.572;
   1:  PR[GP1:91,2] = PR[GP1:90,2] + -10.350;
   1:L PR[91] R[100]mm/sec CNT100;
   1:  PR[GP1:91,1] = PR[GP1:90,1] + -71.914;
   1:  PR[GP1:91,2] = PR[GP1:90,2] + -12.636;
   1:L PR[91] R[100]mm/sec CNT100;
   1:  PR[GP1:91,1] = PR[GP1:90,1] + -70.830;
   1:  PR[GP1:91,2] = PR[GP1:90,2] + -14.784;
   1:L PR[91] R[100]mm/sec CNT100;
   1:  PR[GP1:91,1] = PR[GP1:90,1] + -66.576;
   1:  PR[GP1:91,2] = PR[GP1:90,2] + -21.556;
   1:L PR[91] R[100]mm/sec CNT100;
   1:  PR[GP1:91,1] = PR[GP1:90,1] + -65.111;
   1:  PR[GP1:91,2] = PR[GP1:90,2] + -23.465;
   1:L PR[91] R[100]mm/sec CNT100;
   1:  PR[GP1:91,1] = PR[GP1:90,1] + -63.317;
   1:  PR[GP1:91,2] = PR[GP1:90,2] + -25.069;
   1:L PR[91] R[100]mm/sec CNT100;
   1:  PR[GP1:91,1] = PR[GP1:90,1] + -56.888;
   1:  PR[GP1:91,2] = PR[GP1:90,2] + -29.816;
   1:L PR[91] R[100]mm/sec CNT100;
   1:  PR[GP1:91,1] = PR[GP1:90,1] + -54.827;
   1:  PR[GP1:91,2] = PR[GP1:90,2] + -31.058;
   1:L PR[91] R[100]mm/sec CNT100;
   1:  PR[GP1:91,1] = PR[GP1:90,1] + -52.571;
   1:  PR[GP1:91,2] = PR[GP1:90,2] + -31.896;
   1:L PR[91] R[100]mm/sec CNT100;
   1:  PR[GP1:91,1] = PR[GP1:90,1] + -44.849;
   1:  PR[GP1:91,2] = PR[GP1:90,2] + -33.968;
   1:L PR[91] R[100]mm/sec CNT100;
   1:  PR[GP1:91,1] = PR[GP1:90,1] + -42.477;
   1:  PR[GP1:91,2] = PR[GP1:90,2] + -34.372;
   1:L PR[91] R[100]mm/sec CNT100;
   1:  PR[GP1:91,1] = PR[GP1:90,1] + -40.071;
   1:  PR[GP1:91,2] = PR[GP1:90,2] + -34.328;
   1:L PR[91] R[100]mm/sec CNT100;
   1:  PR[GP1:91,1] = PR[GP1:90,1] + -32.126;
   1:  PR[GP1:91,2] = PR[GP1:90,2] + -33.436;
   1:L PR[91] R[100]mm/sec CNT100;
   1:  PR[GP1:91,1] = PR[GP1:90,1] + -29.770;
   1:  PR[GP1:91,2] = PR[GP1:90,2] + -32.946;
   1:L PR[91] R[100]mm/sec CNT100;
   1:  PR[GP1:91,1] = PR[GP1:90,1] + -27.546;
   1:  PR[GP1:91,2] = PR[GP1:90,2] + -32.026;
   1:L PR[91] R[100]mm/sec CNT100;
   1:  PR[GP1:91,1] = PR[GP1:90,1] + -20.479;
   1:  PR[GP1:91,2] = PR[GP1:90,2] + -28.296;
   1:L PR[91] R[100]mm/sec CNT100;
   1:  PR[GP1:91,1] = PR[GP1:90,1] + -18.465;
   1:  PR[GP1:91,2] = PR[GP1:90,2] + -26.979;
   1:L PR[91] R[100]mm/sec CNT100;
   1:  PR[GP1:91,1] = PR[GP1:90,1] + -16.731;
   1:  PR[GP1:91,2] = PR[GP1:90,2] + -25.311;
   1:L PR[91] R[100]mm/sec CNT100;
   1:  PR[GP1:91,1] = PR[GP1:90,1] + -11.511;
   1:  PR[GP1:91,2] = PR[GP1:90,2] + -19.254;
   1:L PR[91] R[100]mm/sec CNT100;
   1:  PR[GP1:91,1] = PR[GP1:90,1] + -10.117;
   1:  PR[GP1:91,2] = PR[GP1:90,2] + -17.292;
   1:L PR[91] R[100]mm/sec CNT100;
   1:  PR[GP1:91,1] = PR[GP1:90,1] + -9.112;
   1:  PR[GP1:91,2] = PR[GP1:90,2] + -15.106;
   1:L PR[91] R[100]mm/sec CNT100;
   1:  PR[GP1:91,1] = PR[GP1:90,1] + -6.467;
   1:  PR[GP1:91,2] = PR[GP1:90,2] + -7.567;
   1:L PR[91] R[100]mm/sec CNT100;
   1:  PR[GP1:91,1] = PR[GP1:90,1] + -5.853;
   1:  PR[GP1:91,2] = PR[GP1:90,2] + -5.100;
   1:L PR[91] R[100]mm/sec CNT100;
   1:  PR[GP1:91,1] = PR[GP1:90,1] + -4.023;
   1:  PR[GP1:91,2] = PR[GP1:90,2] + -1.796;
   1:L PR[91] R[100]mm/sec CNT100;
   1:  PR[GP1:91,1] = PR[GP1:90,1] + -0.454;
   1:  PR[GP1:91,2] = PR[GP1:90,2] + -0.472;
   1:L PR[91] R[100]mm/sec CNT100;
   1:  PR[GP1:91,1] = PR[GP1:90,1] + 0.667;
   1:L PR[91] R[100]mm/sec CNT100;
   1:  PR[GP1:91,1] = PR[GP1:90,1] + 4.236;
   1:  PR[GP1:91,2] = PR[GP1:90,2] + -1.796;
   1:L PR[91] R[100]mm/sec CNT100;
   1:  PR[GP1:91,1] = PR[GP1:90,1] + 6.052;
   1:  PR[GP1:91,2] = PR[GP1:90,2] + -5.076;
   1:L PR[91] R[100]mm/sec CNT100;
   1:  PR[GP1:91,1] = PR[GP1:90,1] + 8.742;
   1:  PR[GP1:91,2] = PR[GP1:90,2] + -12.742;
   1:L PR[91] R[100]mm/sec CNT100;
   1:  PR[GP1:91,1] = PR[GP1:90,1] + 9.337;
   1:  PR[GP1:91,2] = PR[GP1:90,2] + -15.131;
   1:L PR[91] R[100]mm/sec CNT100;
   1:  PR[GP1:91,1] = PR[GP1:90,1] + 10.319;
   1:  PR[GP1:91,2] = PR[GP1:90,2] + -17.267;
   1:L PR[91] R[100]mm/sec CNT100;
   1:  PR[GP1:91,1] = PR[GP1:90,1] + 15.538;
   1:  PR[GP1:91,2] = PR[GP1:90,2] + -23.323;
   1:L PR[91] R[100]mm/sec CNT100;
   1:  PR[GP1:91,1] = PR[GP1:90,1] + 16.964;
   1:  PR[GP1:91,2] = PR[GP1:90,2] + -25.330;
   1:L PR[91] R[100]mm/sec CNT100;
   1:  PR[GP1:91,1] = PR[GP1:90,1] + 18.658;
   1:  PR[GP1:91,2] = PR[GP1:90,2] + -26.959;
   1:L PR[91] R[100]mm/sec CNT100;
   1:  PR[GP1:91,1] = PR[GP1:90,1] + 25.724;
   1:  PR[GP1:91,2] = PR[GP1:90,2] + -30.690;
   1:L PR[91] R[100]mm/sec CNT100;
   1:  PR[GP1:91,1] = PR[GP1:90,1] + 27.785;
   1:  PR[GP1:91,2] = PR[GP1:90,2] + -32.037;
   1:L PR[91] R[100]mm/sec CNT100;
   1:  PR[GP1:91,1] = PR[GP1:90,1] + 29.957;
   1:  PR[GP1:91,2] = PR[GP1:90,2] + -32.935;
   1:L PR[91] R[100]mm/sec CNT100;
   1:  PR[GP1:91,1] = PR[GP1:90,1] + 37.901;
   1:  PR[GP1:91,2] = PR[GP1:90,2] + -33.827;
   1:L PR[91] R[100]mm/sec CNT100;
   1:  PR[GP1:91,1] = PR[GP1:90,1] + 40.312;
   1:  PR[GP1:91,2] = PR[GP1:90,2] + -34.329;
   1:L PR[91] R[100]mm/sec CNT100;
   1:  PR[GP1:91,1] = PR[GP1:90,1] + 42.662;
   1:  PR[GP1:91,2] = PR[GP1:90,2] + -34.371;
   1:L PR[91] R[100]mm/sec CNT100;
   1:  PR[GP1:91,1] = PR[GP1:90,1] + 50.383;
   1:  PR[GP1:91,2] = PR[GP1:90,2] + -32.300;
   1:L PR[91] R[100]mm/sec CNT100;
   1:  PR[GP1:91,1] = PR[GP1:90,1] + 52.811;
   1:  PR[GP1:91,2] = PR[GP1:90,2] + -31.887;
   1:L PR[91] R[100]mm/sec CNT100;
   1:  PR[GP1:91,1] = PR[GP1:90,1] + 55.014;
   1:  PR[GP1:91,2] = PR[GP1:90,2] + -31.068;
   1:L PR[91] R[100]mm/sec CNT100;
   1:  PR[GP1:91,1] = PR[GP1:90,1] + 61.443;
   1:  PR[GP1:91,2] = PR[GP1:90,2] + -26.322;
   1:L PR[91] R[100]mm/sec CNT100;
   1:  PR[GP1:91,1] = PR[GP1:90,1] + 63.551;
   1:  PR[GP1:91,2] = PR[GP1:90,2] + -25.050;
   1:L PR[91] R[100]mm/sec CNT100;
   1:  PR[GP1:91,1] = PR[GP1:90,1] + 65.303;
   1:  PR[GP1:91,2] = PR[GP1:90,2] + -23.484;
   1:L PR[91] R[100]mm/sec CNT100;
   1:  PR[GP1:91,1] = PR[GP1:90,1] + 69.557;
   1:  PR[GP1:91,2] = PR[GP1:90,2] + -16.713;
   1:L PR[91] R[100]mm/sec CNT100;
   1:  PR[GP1:91,1] = PR[GP1:90,1] + 71.056;
   1:  PR[GP1:91,2] = PR[GP1:90,2] + -14.759;
   1:L PR[91] R[100]mm/sec CNT100;
   1:  PR[GP1:91,1] = PR[GP1:90,1] + 72.114;
   1:  PR[GP1:91,2] = PR[GP1:90,2] + -12.661;
   1:L PR[91] R[100]mm/sec CNT100;
   1:  PR[GP1:91,1] = PR[GP1:90,1] + 73.600;
   1:  PR[GP1:91,2] = PR[GP1:90,2] + -4.806;
   1:L PR[91] R[100]mm/sec CNT100;
   1:  PR[GP1:91,1] = PR[GP1:90,1] + 74.282;
   1:  PR[GP1:91,2] = PR[GP1:90,2] + -2.440;
   1:L PR[91] R[100]mm/sec CNT100;
   1:  PR[GP1:91,1] = PR[GP1:90,1] + 74.501;
   1:  PR[GP1:91,2] = PR[GP1:90,2] + -0.100;
   1:L PR[91] R[100]mm/sec CNT100;
   1:  PR[GP1:91,1] = PR[GP1:90,1] + 73.015;
   1:  PR[GP1:91,2] = PR[GP1:90,2] + 7.754;
   1:L PR[91] R[100]mm/sec CNT100;
   1:  PR[GP1:91,1] = PR[GP1:90,1] + 72.785;
   1:  PR[GP1:91,2] = PR[GP1:90,2] + 10.206;
   1:L PR[91] R[100]mm/sec CNT100;
   1:  PR[GP1:91,1] = PR[GP1:90,1] + 72.127;
   1:  PR[GP1:91,2] = PR[GP1:90,2] + 12.492;
   1:L PR[91] R[100]mm/sec CNT100;
   1:  PR[GP1:91,1] = PR[GP1:90,1] + 71.043;
   1:  PR[GP1:91,2] = PR[GP1:90,2] + 14.640;
   1:L PR[91] R[100]mm/sec CNT100;
   1:  PR[GP1:91,1] = PR[GP1:90,1] + 66.789;
   1:  PR[GP1:91,2] = PR[GP1:90,2] + 21.411;
   1:L PR[91] R[100]mm/sec CNT100;
   1:  PR[GP1:91,1] = PR[GP1:90,1] + 65.324;
   1:  PR[GP1:91,2] = PR[GP1:90,2] + 23.321;
   1:L PR[91] R[100]mm/sec CNT100;
   1:  PR[GP1:91,1] = PR[GP1:90,1] + 63.530;
   1:  PR[GP1:91,2] = PR[GP1:90,2] + 24.925;
   1:L PR[91] R[100]mm/sec CNT100;
   1:  PR[GP1:91,1] = PR[GP1:90,1] + 57.101;
   1:  PR[GP1:91,2] = PR[GP1:90,2] + 29.672;
   1:L PR[91] R[100]mm/sec CNT100;
   1:  PR[GP1:91,1] = PR[GP1:90,1] + 55.040;
   1:  PR[GP1:91,2] = PR[GP1:90,2] + 30.914;
   1:L PR[91] R[100]mm/sec CNT100;
   1:  PR[GP1:91,1] = PR[GP1:90,1] + 52.784;
   1:  PR[GP1:91,2] = PR[GP1:90,2] + 31.752;
   1:L PR[91] R[100]mm/sec CNT100;
   1:  PR[GP1:91,1] = PR[GP1:90,1] + 45.062;
   1:  PR[GP1:91,2] = PR[GP1:90,2] + 33.824;
   1:L PR[91] R[100]mm/sec CNT100;
   1:  PR[GP1:91,1] = PR[GP1:90,1] + 42.690;
   1:  PR[GP1:91,2] = PR[GP1:90,2] + 34.228;
   1:L PR[91] R[100]mm/sec CNT100;
   1:  PR[GP1:91,1] = PR[GP1:90,1] + 40.284;
   1:  PR[GP1:91,2] = PR[GP1:90,2] + 34.184;
   1:L PR[91] R[100]mm/sec CNT100;
   1:  PR[GP1:91,1] = PR[GP1:90,1] + 32.339;
   1:  PR[GP1:91,2] = PR[GP1:90,2] + 33.292;
   1:L PR[91] R[100]mm/sec CNT100;
   1:  PR[GP1:91,1] = PR[GP1:90,1] + 29.983;
   1:  PR[GP1:91,2] = PR[GP1:90,2] + 32.802;
   1:L PR[91] R[100]mm/sec CNT100;
   1:  PR[GP1:91,1] = PR[GP1:90,1] + 27.759;
   1:  PR[GP1:91,2] = PR[GP1:90,2] + 31.882;
   1:L PR[91] R[100]mm/sec CNT100;
   1:  PR[GP1:91,1] = PR[GP1:90,1] + 20.693;
   1:  PR[GP1:91,2] = PR[GP1:90,2] + 28.152;
   1:L PR[91] R[100]mm/sec CNT100;
   1:  PR[GP1:91,1] = PR[GP1:90,1] + 18.678;
   1:  PR[GP1:91,2] = PR[GP1:90,2] + 26.835;
   1:L PR[91] R[100]mm/sec CNT100;
   1:  PR[GP1:91,1] = PR[GP1:90,1] + 16.944;
   1:  PR[GP1:91,2] = PR[GP1:90,2] + 25.167;
   1:L PR[91] R[100]mm/sec CNT100;
   1:  PR[GP1:91,1] = PR[GP1:90,1] + 11.725;
   1:  PR[GP1:91,2] = PR[GP1:90,2] + 19.110;
   1:L PR[91] R[100]mm/sec CNT100;
   1:  PR[GP1:91,1] = PR[GP1:90,1] + 10.330;
   1:  PR[GP1:91,2] = PR[GP1:90,2] + 17.148;
   1:L PR[91] R[100]mm/sec CNT100;
   1:  PR[GP1:91,1] = PR[GP1:90,1] + 9.325;
   1:  PR[GP1:91,2] = PR[GP1:90,2] + 14.962;
   1:L PR[91] R[100]mm/sec CNT100;
   1:  PR[GP1:91,1] = PR[GP1:90,1] + 6.680;
   1:  PR[GP1:91,2] = PR[GP1:90,2] + 7.423;
   1:L PR[91] R[100]mm/sec CNT100;
   1:  PR[GP1:91,1] = PR[GP1:90,1] + 6.066;
   1:  PR[GP1:91,2] = PR[GP1:90,2] + 4.956;
   1:L PR[91] R[100]mm/sec CNT100;
   1:  PR[GP1:91,1] = PR[GP1:90,1] + 4.236;
   1:  PR[GP1:91,2] = PR[GP1:90,2] + 1.652;
   1:L PR[91] R[100]mm/sec CNT100;
   1:  PR[GP1:91,1] = PR[GP1:90,1] + 0.667;
   1:  PR[GP1:91,2] = PR[GP1:90,2] + 0.328;
   1:L PR[91] R[100]mm/sec CNT100;
   1:  PR[GP1:91,1] = PR[GP1:90,1] + -0.454;
   1:L PR[91] R[100]mm/sec CNT100;
   1:  ! -- Layer/Ebene 6 -- !;
   1:  PR[91] = PR[90];
   1:  PR[GP1:91,1] = PR[GP1:90,1] + -4.023;
   1:  PR[GP1:91,2] = PR[GP1:90,2] + 1.652;
   1:  PR[GP1:91,3] = PR[GP1:90,3] + 3.965;
   1:L PR[91] R[100]mm/sec CNT100;
   1:  PR[GP1:91,1] = PR[GP1:90,1] + -5.839;
   1:  PR[GP1:91,2] = PR[GP1:90,2] + 4.932;
   1:L PR[91] R[100]mm/sec CNT100;
   1:  PR[GP1:91,1] = PR[GP1:90,1] + -8.200;
   1:  PR[GP1:91,2] = PR[GP1:90,2] + 11.662;
   1:L PR[91] R[100]mm/sec CNT100;
   1:  PR[GP1:91,1] = PR[GP1:90,1] + -8.916;
   1:  PR[GP1:91,2] = PR[GP1:90,2] + 14.535;
   1:L PR[91] R[100]mm/sec CNT100;
   1:  PR[GP1:91,1] = PR[GP1:90,1] + -10.106;
   1:  PR[GP1:91,2] = PR[GP1:90,2] + 17.123;
   1:L PR[91] R[100]mm/sec CNT100;
   1:  PR[GP1:91,1] = PR[GP1:90,1] + -14.677;
   1:  PR[GP1:91,2] = PR[GP1:90,2] + 22.428;
   1:L PR[91] R[100]mm/sec CNT100;
   1:  PR[GP1:91,1] = PR[GP1:90,1] + -16.392;
   1:  PR[GP1:91,2] = PR[GP1:90,2] + 24.841;
   1:L PR[91] R[100]mm/sec CNT100;
   1:  PR[GP1:91,1] = PR[GP1:90,1] + -18.445;
   1:  PR[GP1:91,2] = PR[GP1:90,2] + 26.816;
   1:L PR[91] R[100]mm/sec CNT100;
   1:  PR[GP1:91,1] = PR[GP1:90,1] + -24.634;
   1:  PR[GP1:91,2] = PR[GP1:90,2] + 30.083;
   1:L PR[91] R[100]mm/sec CNT100;
   1:  PR[GP1:91,1] = PR[GP1:90,1] + -27.112;
   1:  PR[GP1:91,2] = PR[GP1:90,2] + 31.703;
   1:L PR[91] R[100]mm/sec CNT100;
   1:  PR[GP1:91,1] = PR[GP1:90,1] + -29.744;
   1:  PR[GP1:91,2] = PR[GP1:90,2] + 32.791;
   1:L PR[91] R[100]mm/sec CNT100;
   1:  PR[GP1:91,1] = PR[GP1:90,1] + -36.703;
   1:  PR[GP1:91,2] = PR[GP1:90,2] + 33.573;
   1:L PR[91] R[100]mm/sec CNT100;
   1:  PR[GP1:91,1] = PR[GP1:90,1] + -39.601;
   1:  PR[GP1:91,2] = PR[GP1:90,2] + 34.176;
   1:L PR[91] R[100]mm/sec CNT100;
   1:  PR[GP1:91,1] = PR[GP1:90,1] + -42.449;
   1:  PR[GP1:91,2] = PR[GP1:90,2] + 34.227;
   1:L PR[91] R[100]mm/sec CNT100;
   1:  PR[GP1:91,1] = PR[GP1:90,1] + -49.212;
   1:  PR[GP1:91,2] = PR[GP1:90,2] + 32.413;
   1:L PR[91] R[100]mm/sec CNT100;
   1:  PR[GP1:91,1] = PR[GP1:90,1] + -52.131;
   1:  PR[GP1:91,2] = PR[GP1:90,2] + 31.916;
   1:L PR[91] R[100]mm/sec CNT100;
   1:  PR[GP1:91,1] = PR[GP1:90,1] + -54.801;
   1:  PR[GP1:91,2] = PR[GP1:90,2] + 30.924;
   1:L PR[91] R[100]mm/sec CNT100;
   1:  PR[GP1:91,1] = PR[GP1:90,1] + -60.432;
   1:  PR[GP1:91,2] = PR[GP1:90,2] + 26.767;
   1:L PR[91] R[100]mm/sec CNT100;
   1:  PR[GP1:91,1] = PR[GP1:90,1] + -62.967;
   1:  PR[GP1:91,2] = PR[GP1:90,2] + 25.238;
   1:L PR[91] R[100]mm/sec CNT100;
   1:  PR[GP1:91,1] = PR[GP1:90,1] + -65.090;
   1:  PR[GP1:91,2] = PR[GP1:90,2] + 23.340;
   1:L PR[91] R[100]mm/sec CNT100;
   1:  PR[GP1:91,1] = PR[GP1:90,1] + -68.816;
   1:  PR[GP1:91,2] = PR[GP1:90,2] + 17.409;
   1:L PR[91] R[100]mm/sec CNT100;
   1:  PR[GP1:91,1] = PR[GP1:90,1] + -70.618;
   1:  PR[GP1:91,2] = PR[GP1:90,2] + 15.060;
   1:L PR[91] R[100]mm/sec CNT100;
   1:  PR[GP1:91,1] = PR[GP1:90,1] + -71.901;
   1:  PR[GP1:91,2] = PR[GP1:90,2] + 12.517;
   1:L PR[91] R[100]mm/sec CNT100;
   1:  PR[GP1:91,1] = PR[GP1:90,1] + -73.203;
   1:  PR[GP1:91,2] = PR[GP1:90,2] + 5.637;
   1:L PR[91] R[100]mm/sec CNT100;
   1:  PR[GP1:91,1] = PR[GP1:90,1] + -74.022;
   1:  PR[GP1:91,2] = PR[GP1:90,2] + 2.792;
   1:L PR[91] R[100]mm/sec CNT100;
   1:  PR[GP1:91,1] = PR[GP1:90,1] + -74.288;
   1:  PR[GP1:91,2] = PR[GP1:90,2] + -0.044;
   1:L PR[91] R[100]mm/sec CNT100;
   1:  PR[GP1:91,1] = PR[GP1:90,1] + -72.986;
   1:  PR[GP1:91,2] = PR[GP1:90,2] + -6.924;
   1:L PR[91] R[100]mm/sec CNT100;
   1:  PR[GP1:91,1] = PR[GP1:90,1] + -72.710;
   1:  PR[GP1:91,2] = PR[GP1:90,2] + -9.871;
   1:L PR[91] R[100]mm/sec CNT100;
   1:  PR[GP1:91,1] = PR[GP1:90,1] + -71.914;
   1:  PR[GP1:91,2] = PR[GP1:90,2] + -12.636;
   1:L PR[91] R[100]mm/sec CNT100;
   1:  PR[GP1:91,1] = PR[GP1:90,1] + -70.605;
   1:  PR[GP1:91,2] = PR[GP1:90,2] + -15.229;
   1:L PR[91] R[100]mm/sec CNT100;
   1:  PR[GP1:91,1] = PR[GP1:90,1] + -66.879;
   1:  PR[GP1:91,2] = PR[GP1:90,2] + -21.160;
   1:L PR[91] R[100]mm/sec CNT100;
   1:  PR[GP1:91,1] = PR[GP1:90,1] + -65.111;
   1:  PR[GP1:91,2] = PR[GP1:90,2] + -23.465;
   1:L PR[91] R[100]mm/sec CNT100;
   1:  PR[GP1:91,1] = PR[GP1:90,1] + -62.946;
   1:  PR[GP1:91,2] = PR[GP1:90,2] + -25.401;
   1:L PR[91] R[100]mm/sec CNT100;
   1:  PR[GP1:91,1] = PR[GP1:90,1] + -57.315;
   1:  PR[GP1:91,2] = PR[GP1:90,2] + -29.558;
   1:L PR[91] R[100]mm/sec CNT100;
   1:  PR[GP1:91,1] = PR[GP1:90,1] + -54.827;
   1:  PR[GP1:91,2] = PR[GP1:90,2] + -31.058;
   1:L PR[91] R[100]mm/sec CNT100;
   1:  PR[GP1:91,1] = PR[GP1:90,1] + -52.105;
   1:  PR[GP1:91,2] = PR[GP1:90,2] + -32.070;
   1:L PR[91] R[100]mm/sec CNT100;
   1:  PR[GP1:91,1] = PR[GP1:90,1] + -45.341;
   1:  PR[GP1:91,2] = PR[GP1:90,2] + -33.884;
   1:L PR[91] R[100]mm/sec CNT100;
   1:  PR[GP1:91,1] = PR[GP1:90,1] + -42.477;
   1:  PR[GP1:91,2] = PR[GP1:90,2] + -34.372;
   1:L PR[91] R[100]mm/sec CNT100;
   1:  PR[GP1:91,1] = PR[GP1:90,1] + -39.573;
   1:  PR[GP1:91,2] = PR[GP1:90,2] + -34.319;
   1:L PR[91] R[100]mm/sec CNT100;
   1:  PR[GP1:91,1] = PR[GP1:90,1] + -32.614;
   1:  PR[GP1:91,2] = PR[GP1:90,2] + -33.538;
   1:L PR[91] R[100]mm/sec CNT100;
   1:  PR[GP1:91,1] = PR[GP1:90,1] + -29.771;
   1:  PR[GP1:91,2] = PR[GP1:90,2] + -32.946;
   1:L PR[91] R[100]mm/sec CNT100;
   1:  PR[GP1:91,1] = PR[GP1:90,1] + -27.086;
   1:  PR[GP1:91,2] = PR[GP1:90,2] + -31.836;
   1:L PR[91] R[100]mm/sec CNT100;
   1:  PR[GP1:91,1] = PR[GP1:90,1] + -20.896;
   1:  PR[GP1:91,2] = PR[GP1:90,2] + -28.569;
   1:L PR[91] R[100]mm/sec CNT100;
   1:  PR[GP1:91,1] = PR[GP1:90,1] + -18.465;
   1:  PR[GP1:91,2] = PR[GP1:90,2] + -26.979;
   1:L PR[91] R[100]mm/sec CNT100;
   1:  PR[GP1:91,1] = PR[GP1:90,1] + -16.372;
   1:  PR[GP1:91,2] = PR[GP1:90,2] + -24.966;
   1:L PR[91] R[100]mm/sec CNT100;
   1:  PR[GP1:91,1] = PR[GP1:90,1] + -11.800;
   1:  PR[GP1:91,2] = PR[GP1:90,2] + -19.660;
   1:L PR[91] R[100]mm/sec CNT100;
   1:  PR[GP1:91,1] = PR[GP1:90,1] + -10.117;
   1:  PR[GP1:91,2] = PR[GP1:90,2] + -17.293;
   1:L PR[91] R[100]mm/sec CNT100;
   1:  PR[GP1:91,1] = PR[GP1:90,1] + -8.904;
   1:  PR[GP1:91,2] = PR[GP1:90,2] + -14.654;
   1:L PR[91] R[100]mm/sec CNT100;
   1:  PR[GP1:91,1] = PR[GP1:90,1] + -6.587;
   1:  PR[GP1:91,2] = PR[GP1:90,2] + -8.050;
   1:L PR[91] R[100]mm/sec CNT100;
   1:  PR[GP1:91,1] = PR[GP1:90,1] + -5.853;
   1:  PR[GP1:91,2] = PR[GP1:90,2] + -5.100;
   1:L PR[91] R[100]mm/sec CNT100;
   1:  PR[GP1:91,1] = PR[GP1:90,1] + -4.023;
   1:  PR[GP1:91,2] = PR[GP1:90,2] + -1.796;
   1:L PR[91] R[100]mm/sec CNT100;
   1:  PR[GP1:91,1] = PR[GP1:90,1] + -0.454;
   1:  PR[GP1:91,2] = PR[GP1:90,2] + -0.472;
   1:L PR[91] R[100]mm/sec CNT100;
   1:  PR[GP1:91,1] = PR[GP1:90,1] + 0.667;
   1:L PR[91] R[100]mm/sec CNT100;
   1:  PR[GP1:91,1] = PR[GP1:90,1] + 4.236;
   1:  PR[GP1:91,2] = PR[GP1:90,2] + -1.796;
   1:L PR[91] R[100]mm/sec CNT100;
   1:  PR[GP1:91,1] = PR[GP1:90,1] + 6.052;
   1:  PR[GP1:91,2] = PR[GP1:90,2] + -5.076;
   1:L PR[91] R[100]mm/sec CNT100;
   1:  PR[GP1:91,1] = PR[GP1:90,1] + 8.414;
   1:  PR[GP1:91,2] = PR[GP1:90,2] + -11.806;
   1:L PR[91] R[100]mm/sec CNT100;
   1:  PR[GP1:91,1] = PR[GP1:90,1] + 9.129;
   1:  PR[GP1:91,2] = PR[GP1:90,2] + -14.679;
   1:L PR[91] R[100]mm/sec CNT100;
   1:  PR[GP1:91,1] = PR[GP1:90,1] + 10.319;
   1:  PR[GP1:91,2] = PR[GP1:90,2] + -17.267;
   1:L PR[91] R[100]mm/sec CNT100;
   1:  PR[GP1:91,1] = PR[GP1:90,1] + 14.890;
   1:  PR[GP1:91,2] = PR[GP1:90,2] + -22.572;
   1:L PR[91] R[100]mm/sec CNT100;
   1:  PR[GP1:91,1] = PR[GP1:90,1] + 16.605;
   1:  PR[GP1:91,2] = PR[GP1:90,2] + -24.985;
   1:L PR[91] R[100]mm/sec CNT100;
   1:  PR[GP1:91,1] = PR[GP1:90,1] + 18.658;
   1:  PR[GP1:91,2] = PR[GP1:90,2] + -26.960;
   1:L PR[91] R[100]mm/sec CNT100;
   1:  PR[GP1:91,1] = PR[GP1:90,1] + 24.847;
   1:  PR[GP1:91,2] = PR[GP1:90,2] + -30.227;
   1:L PR[91] R[100]mm/sec CNT100;
   1:  PR[GP1:91,1] = PR[GP1:90,1] + 27.326;
   1:  PR[GP1:91,2] = PR[GP1:90,2] + -31.847;
   1:L PR[91] R[100]mm/sec CNT100;
   1:  PR[GP1:91,1] = PR[GP1:90,1] + 29.958;
   1:  PR[GP1:91,2] = PR[GP1:90,2] + -32.935;
   1:L PR[91] R[100]mm/sec CNT100;
   1:  PR[GP1:91,1] = PR[GP1:90,1] + 36.916;
   1:  PR[GP1:91,2] = PR[GP1:90,2] + -33.717;
   1:L PR[91] R[100]mm/sec CNT100;
   1:  PR[GP1:91,1] = PR[GP1:90,1] + 39.815;
   1:  PR[GP1:91,2] = PR[GP1:90,2] + -34.320;
   1:L PR[91] R[100]mm/sec CNT100;
   1:  PR[GP1:91,1] = PR[GP1:90,1] + 42.662;
   1:  PR[GP1:91,2] = PR[GP1:90,2] + -34.371;
   1:L PR[91] R[100]mm/sec CNT100;
   1:  PR[GP1:91,1] = PR[GP1:90,1] + 49.425;
   1:  PR[GP1:91,2] = PR[GP1:90,2] + -32.557;
   1:L PR[91] R[100]mm/sec CNT100;
   1:  PR[GP1:91,1] = PR[GP1:90,1] + 52.344;
   1:  PR[GP1:91,2] = PR[GP1:90,2] + -32.060;
   1:L PR[91] R[100]mm/sec CNT100;
   1:  PR[GP1:91,1] = PR[GP1:90,1] + 55.014;
   1:  PR[GP1:91,2] = PR[GP1:90,2] + -31.068;
   1:L PR[91] R[100]mm/sec CNT100;
   1:  PR[GP1:91,1] = PR[GP1:90,1] + 60.645;
   1:  PR[GP1:91,2] = PR[GP1:90,2] + -26.911;
   1:L PR[91] R[100]mm/sec CNT100;
   1:  PR[GP1:91,1] = PR[GP1:90,1] + 63.180;
   1:  PR[GP1:91,2] = PR[GP1:90,2] + -25.382;
   1:L PR[91] R[100]mm/sec CNT100;
   1:  PR[GP1:91,1] = PR[GP1:90,1] + 65.303;
   1:  PR[GP1:91,2] = PR[GP1:90,2] + -23.484;
   1:L PR[91] R[100]mm/sec CNT100;
   1:  PR[GP1:91,1] = PR[GP1:90,1] + 69.029;
   1:  PR[GP1:91,2] = PR[GP1:90,2] + -17.553;
   1:L PR[91] R[100]mm/sec CNT100;
   1:  PR[GP1:91,1] = PR[GP1:90,1] + 70.831;
   1:  PR[GP1:91,2] = PR[GP1:90,2] + -15.204;
   1:L PR[91] R[100]mm/sec CNT100;
   1:  PR[GP1:91,1] = PR[GP1:90,1] + 72.114;
   1:  PR[GP1:91,2] = PR[GP1:90,2] + -12.661;
   1:L PR[91] R[100]mm/sec CNT100;
   1:  PR[GP1:91,1] = PR[GP1:90,1] + 73.416;
   1:  PR[GP1:91,2] = PR[GP1:90,2] + -5.781;
   1:L PR[91] R[100]mm/sec CNT100;
   1:  PR[GP1:91,1] = PR[GP1:90,1] + 74.236;
   1:  PR[GP1:91,2] = PR[GP1:90,2] + -2.936;
   1:L PR[91] R[100]mm/sec CNT100;
   1:  PR[GP1:91,1] = PR[GP1:90,1] + 74.501;
   1:  PR[GP1:91,2] = PR[GP1:90,2] + -0.100;
   1:L PR[91] R[100]mm/sec CNT100;
   1:  PR[GP1:91,1] = PR[GP1:90,1] + 73.200;
   1:  PR[GP1:91,2] = PR[GP1:90,2] + 6.780;
   1:L PR[91] R[100]mm/sec CNT100;
   1:  PR[GP1:91,1] = PR[GP1:90,1] + 72.923;
   1:  PR[GP1:91,2] = PR[GP1:90,2] + 9.727;
   1:L PR[91] R[100]mm/sec CNT100;
   1:  PR[GP1:91,1] = PR[GP1:90,1] + 72.127;
   1:  PR[GP1:91,2] = PR[GP1:90,2] + 12.492;
   1:L PR[91] R[100]mm/sec CNT100;
   1:  PR[GP1:91,1] = PR[GP1:90,1] + 70.819;
   1:  PR[GP1:91,2] = PR[GP1:90,2] + 15.085;
   1:L PR[91] R[100]mm/sec CNT100;
   1:  PR[GP1:91,1] = PR[GP1:90,1] + 67.092;
   1:  PR[GP1:91,2] = PR[GP1:90,2] + 21.016;
   1:L PR[91] R[100]mm/sec CNT100;
   1:  PR[GP1:91,1] = PR[GP1:90,1] + 65.325;
   1:  PR[GP1:91,2] = PR[GP1:90,2] + 23.321;
   1:L PR[91] R[100]mm/sec CNT100;
   1:  PR[GP1:91,1] = PR[GP1:90,1] + 63.159;
   1:  PR[GP1:91,2] = PR[GP1:90,2] + 25.257;
   1:L PR[91] R[100]mm/sec CNT100;
   1:  PR[GP1:91,1] = PR[GP1:90,1] + 57.528;
   1:  PR[GP1:91,2] = PR[GP1:90,2] + 29.414;
   1:L PR[91] R[100]mm/sec CNT100;
   1:  PR[GP1:91,1] = PR[GP1:90,1] + 55.040;
   1:  PR[GP1:91,2] = PR[GP1:90,2] + 30.914;
   1:L PR[91] R[100]mm/sec CNT100;
   1:  PR[GP1:91,1] = PR[GP1:90,1] + 52.318;
   1:  PR[GP1:91,2] = PR[GP1:90,2] + 31.926;
   1:L PR[91] R[100]mm/sec CNT100;
   1:  PR[GP1:91,1] = PR[GP1:90,1] + 45.554;
   1:  PR[GP1:91,2] = PR[GP1:90,2] + 33.740;
   1:L PR[91] R[100]mm/sec CNT100;
   1:  PR[GP1:91,1] = PR[GP1:90,1] + 42.691;
   1:  PR[GP1:91,2] = PR[GP1:90,2] + 34.228;
   1:L PR[91] R[100]mm/sec CNT100;
   1:  PR[GP1:91,1] = PR[GP1:90,1] + 39.786;
   1:  PR[GP1:91,2] = PR[GP1:90,2] + 34.175;
   1:L PR[91] R[100]mm/sec CNT100;
   1:  PR[GP1:91,1] = PR[GP1:90,1] + 32.828;
   1:  PR[GP1:91,2] = PR[GP1:90,2] + 33.394;
   1:L PR[91] R[100]mm/sec CNT100;
   1:  PR[GP1:91,1] = PR[GP1:90,1] + 29.984;
   1:  PR[GP1:91,2] = PR[GP1:90,2] + 32.802;
   1:L PR[91] R[100]mm/sec CNT100;
   1:  PR[GP1:91,1] = PR[GP1:90,1] + 27.300;
   1:  PR[GP1:91,2] = PR[GP1:90,2] + 31.692;
   1:L PR[91] R[100]mm/sec CNT100;
   1:  PR[GP1:91,1] = PR[GP1:90,1] + 21.110;
   1:  PR[GP1:91,2] = PR[GP1:90,2] + 28.425;
   1:L PR[91] R[100]mm/sec CNT100;
   1:  PR[GP1:91,1] = PR[GP1:90,1] + 18.678;
   1:  PR[GP1:91,2] = PR[GP1:90,2] + 26.835;
   1:L PR[91] R[100]mm/sec CNT100;
   1:  PR[GP1:91,1] = PR[GP1:90,1] + 16.585;
   1:  PR[GP1:91,2] = PR[GP1:90,2] + 24.822;
   1:L PR[91] R[100]mm/sec CNT100;
   1:  PR[GP1:91,1] = PR[GP1:90,1] + 12.013;
   1:  PR[GP1:91,2] = PR[GP1:90,2] + 19.516;
   1:L PR[91] R[100]mm/sec CNT100;
   1:  PR[GP1:91,1] = PR[GP1:90,1] + 10.331;
   1:  PR[GP1:91,2] = PR[GP1:90,2] + 17.149;
   1:L PR[91] R[100]mm/sec CNT100;
   1:  PR[GP1:91,1] = PR[GP1:90,1] + 9.117;
   1:  PR[GP1:91,2] = PR[GP1:90,2] + 14.510;
   1:L PR[91] R[100]mm/sec CNT100;
   1:  PR[GP1:91,1] = PR[GP1:90,1] + 6.800;
   1:  PR[GP1:91,2] = PR[GP1:90,2] + 7.906;
   1:L PR[91] R[100]mm/sec CNT100;
   1:  PR[GP1:91,1] = PR[GP1:90,1] + 6.066;
   1:  PR[GP1:91,2] = PR[GP1:90,2] + 4.956;
   1:L PR[91] R[100]mm/sec CNT100;
   1:  PR[GP1:91,1] = PR[GP1:90,1] + 4.236;
   1:  PR[GP1:91,2] = PR[GP1:90,2] + 1.652;
   1:L PR[91] R[100]mm/sec CNT100;
   1:  PR[GP1:91,1] = PR[GP1:90,1] + 0.667;
   1:  PR[GP1:91,2] = PR[GP1:90,2] + 0.328;
   1:L PR[91] R[100]mm/sec CNT100;
   1:  PR[GP1:91,1] = PR[GP1:90,1] + -0.454;
   1:L PR[91] R[100]mm/sec CNT100;
   1:  ! -- Layer/Ebene 7 -- !;
   1:  PR[91] = PR[90];
   1:  PR[GP1:91,1] = PR[GP1:90,1] + -4.023;
   1:  PR[GP1:91,2] = PR[GP1:90,2] + 1.652;
   1:  PR[GP1:91,3] = PR[GP1:90,3] + 4.575;
   1:L PR[91] R[100]mm/sec CNT100;
   1:  PR[GP1:91,1] = PR[GP1:90,1] + -5.839;
   1:  PR[GP1:91,2] = PR[GP1:90,2] + 4.932;
   1:L PR[91] R[100]mm/sec CNT100;
   1:  PR[GP1:91,1] = PR[GP1:90,1] + -7.872;
   1:  PR[GP1:91,2] = PR[GP1:90,2] + 10.727;
   1:L PR[91] R[100]mm/sec CNT100;
   1:  PR[GP1:91,1] = PR[GP1:90,1] + -8.708;
   1:  PR[GP1:91,2] = PR[GP1:90,2] + 14.083;
   1:L PR[91] R[100]mm/sec CNT100;
   1:  PR[GP1:91,1] = PR[GP1:90,1] + -10.106;
   1:  PR[GP1:91,2] = PR[GP1:90,2] + 17.123;
   1:L PR[91] R[100]mm/sec CNT100;
   1:  PR[GP1:91,1] = PR[GP1:90,1] + -14.029;
   1:  PR[GP1:91,2] = PR[GP1:90,2] + 21.677;
   1:L PR[91] R[100]mm/sec CNT100;
   1:  PR[GP1:91,1] = PR[GP1:90,1] + -16.033;
   1:  PR[GP1:91,2] = PR[GP1:90,2] + 24.496;
   1:L PR[91] R[100]mm/sec CNT100;
   1:  PR[GP1:91,1] = PR[GP1:90,1] + -18.445;
   1:  PR[GP1:91,2] = PR[GP1:90,2] + 26.816;
   1:L PR[91] R[100]mm/sec CNT100;
   1:  PR[GP1:91,1] = PR[GP1:90,1] + -23.757;
   1:  PR[GP1:91,2] = PR[GP1:90,2] + 29.620;
   1:L PR[91] R[100]mm/sec CNT100;
   1:  PR[GP1:91,1] = PR[GP1:90,1] + -26.653;
   1:  PR[GP1:91,2] = PR[GP1:90,2] + 31.513;
   1:L PR[91] R[100]mm/sec CNT100;
   1:  PR[GP1:91,1] = PR[GP1:90,1] + -29.745;
   1:  PR[GP1:91,2] = PR[GP1:90,2] + 32.791;
   1:L PR[91] R[100]mm/sec CNT100;
   1:  PR[GP1:91,1] = PR[GP1:90,1] + -35.717;
   1:  PR[GP1:91,2] = PR[GP1:90,2] + 33.462;
   1:L PR[91] R[100]mm/sec CNT100;
   1:  PR[GP1:91,1] = PR[GP1:90,1] + -39.104;
   1:  PR[GP1:91,2] = PR[GP1:90,2] + 34.167;
   1:L PR[91] R[100]mm/sec CNT100;
   1:  PR[GP1:91,1] = PR[GP1:90,1] + -42.449;
   1:  PR[GP1:91,2] = PR[GP1:90,2] + 34.227;
   1:L PR[91] R[100]mm/sec CNT100;
   1:  PR[GP1:91,1] = PR[GP1:90,1] + -48.254;
   1:  PR[GP1:91,2] = PR[GP1:90,2] + 32.670;
   1:L PR[91] R[100]mm/sec CNT100;
   1:  PR[GP1:91,1] = PR[GP1:90,1] + -51.664;
   1:  PR[GP1:91,2] = PR[GP1:90,2] + 32.089;
   1:L PR[91] R[100]mm/sec CNT100;
   1:  PR[GP1:91,1] = PR[GP1:90,1] + -54.801;
   1:  PR[GP1:91,2] = PR[GP1:90,2] + 30.924;
   1:L PR[91] R[100]mm/sec CNT100;
   1:  PR[GP1:91,1] = PR[GP1:90,1] + -59.634;
   1:  PR[GP1:91,2] = PR[GP1:90,2] + 27.356;
   1:L PR[91] R[100]mm/sec CNT100;
   1:  PR[GP1:91,1] = PR[GP1:90,1] + -62.596;
   1:  PR[GP1:91,2] = PR[GP1:90,2] + 25.570;
   1:L PR[91] R[100]mm/sec CNT100;
   1:  PR[GP1:91,1] = PR[GP1:90,1] + -65.091;
   1:  PR[GP1:91,2] = PR[GP1:90,2] + 23.339;
   1:L PR[91] R[100]mm/sec CNT100;
   1:  PR[GP1:91,1] = PR[GP1:90,1] + -68.289;
   1:  PR[GP1:91,2] = PR[GP1:90,2] + 18.249;
   1:L PR[91] R[100]mm/sec CNT100;
   1:  PR[GP1:91,1] = PR[GP1:90,1] + -70.394;
   1:  PR[GP1:91,2] = PR[GP1:90,2] + 15.504;
   1:L PR[91] R[100]mm/sec CNT100;
   1:  PR[GP1:91,1] = PR[GP1:90,1] + -71.901;
   1:  PR[GP1:91,2] = PR[GP1:90,2] + 12.517;
   1:L PR[91] R[100]mm/sec CNT100;
   1:  PR[GP1:91,1] = PR[GP1:90,1] + -73.019;
   1:  PR[GP1:91,2] = PR[GP1:90,2] + 6.612;
   1:L PR[91] R[100]mm/sec CNT100;
   1:  PR[GP1:91,1] = PR[GP1:90,1] + -73.976;
   1:  PR[GP1:91,2] = PR[GP1:90,2] + 3.288;
   1:L PR[91] R[100]mm/sec CNT100;
   1:  PR[GP1:91,1] = PR[GP1:90,1] + -74.288;
   1:  PR[GP1:91,2] = PR[GP1:90,2] + -0.044;
   1:L PR[91] R[100]mm/sec CNT100;
   1:  PR[GP1:91,1] = PR[GP1:90,1] + -73.171;
   1:  PR[GP1:91,2] = PR[GP1:90,2] + -5.949;
   1:L PR[91] R[100]mm/sec CNT100;
   1:  PR[GP1:91,1] = PR[GP1:90,1] + -72.848;
   1:  PR[GP1:91,2] = PR[GP1:90,2] + -9.393;
   1:L PR[91] R[100]mm/sec CNT100;
   1:  PR[GP1:91,1] = PR[GP1:90,1] + -71.914;
   1:  PR[GP1:91,2] = PR[GP1:90,2] + -12.636;
   1:L PR[91] R[100]mm/sec CNT100;
   1:  PR[GP1:91,1] = PR[GP1:90,1] + -70.381;
   1:  PR[GP1:91,2] = PR[GP1:90,2] + -15.673;
   1:L PR[91] R[100]mm/sec CNT100;
   1:  PR[GP1:91,1] = PR[GP1:90,1] + -67.183;
   1:  PR[GP1:91,2] = PR[GP1:90,2] + -20.764;
   1:L PR[91] R[100]mm/sec CNT100;
   1:  PR[GP1:91,1] = PR[GP1:90,1] + -65.112;
   1:  PR[GP1:91,2] = PR[GP1:90,2] + -23.464;
   1:L PR[91] R[100]mm/sec CNT100;
   1:  PR[GP1:91,1] = PR[GP1:90,1] + -62.575;
   1:  PR[GP1:91,2] = PR[GP1:90,2] + -25.732;
   1:L PR[91] R[100]mm/sec CNT100;
   1:  PR[GP1:91,1] = PR[GP1:90,1] + -57.742;
   1:  PR[GP1:91,2] = PR[GP1:90,2] + -29.301;
   1:L PR[91] R[100]mm/sec CNT100;
   1:  PR[GP1:91,1] = PR[GP1:90,1] + -54.827;
   1:  PR[GP1:91,2] = PR[GP1:90,2] + -31.058;
   1:L PR[91] R[100]mm/sec CNT100;
   1:  PR[GP1:91,1] = PR[GP1:90,1] + -51.638;
   1:  PR[GP1:91,2] = PR[GP1:90,2] + -32.243;
   1:L PR[91] R[100]mm/sec CNT100;
   1:  PR[GP1:91,1] = PR[GP1:90,1] + -45.832;
   1:  PR[GP1:91,2] = PR[GP1:90,2] + -33.800;
   1:L PR[91] R[100]mm/sec CNT100;
   1:  PR[GP1:91,1] = PR[GP1:90,1] + -42.478;
   1:  PR[GP1:91,2] = PR[GP1:90,2] + -34.372;
   1:L PR[91] R[100]mm/sec CNT100;
   1:  PR[GP1:91,1] = PR[GP1:90,1] + -39.076;
   1:  PR[GP1:91,2] = PR[GP1:90,2] + -34.310;
   1:L PR[91] R[100]mm/sec CNT100;
   1:  PR[GP1:91,1] = PR[GP1:90,1] + -33.103;
   1:  PR[GP1:91,2] = PR[GP1:90,2] + -33.639;
   1:L PR[91] R[100]mm/sec CNT100;
   1:  PR[GP1:91,1] = PR[GP1:90,1] + -29.771;
   1:  PR[GP1:91,2] = PR[GP1:90,2] + -32.946;
   1:L PR[91] R[100]mm/sec CNT100;
   1:  PR[GP1:91,1] = PR[GP1:90,1] + -26.627;
   1:  PR[GP1:91,2] = PR[GP1:90,2] + -31.646;
   1:L PR[91] R[100]mm/sec CNT100;
   1:  PR[GP1:91,1] = PR[GP1:90,1] + -21.314;
   1:  PR[GP1:91,2] = PR[GP1:90,2] + -28.841;
   1:L PR[91] R[100]mm/sec CNT100;
   1:  PR[GP1:91,1] = PR[GP1:90,1] + -18.465;
   1:  PR[GP1:91,2] = PR[GP1:90,2] + -26.979;
   1:L PR[91] R[100]mm/sec CNT100;
   1:  PR[GP1:91,1] = PR[GP1:90,1] + -16.013;
   1:  PR[GP1:91,2] = PR[GP1:90,2] + -24.621;
   1:L PR[91] R[100]mm/sec CNT100;
   1:  PR[GP1:91,1] = PR[GP1:90,1] + -12.089;
   1:  PR[GP1:91,2] = PR[GP1:90,2] + -20.067;
   1:L PR[91] R[100]mm/sec CNT100;
   1:  PR[GP1:91,1] = PR[GP1:90,1] + -10.118;
   1:  PR[GP1:91,2] = PR[GP1:90,2] + -17.293;
   1:L PR[91] R[100]mm/sec CNT100;
   1:  PR[GP1:91,1] = PR[GP1:90,1] + -8.696;
   1:  PR[GP1:91,2] = PR[GP1:90,2] + -14.202;
   1:L PR[91] R[100]mm/sec CNT100;
   1:  PR[GP1:91,1] = PR[GP1:90,1] + -6.707;
   1:  PR[GP1:91,2] = PR[GP1:90,2] + -8.534;
   1:L PR[91] R[100]mm/sec CNT100;
   1:  PR[GP1:91,1] = PR[GP1:90,1] + -5.853;
   1:  PR[GP1:91,2] = PR[GP1:90,2] + -5.100;
   1:L PR[91] R[100]mm/sec CNT100;
   1:  PR[GP1:91,1] = PR[GP1:90,1] + -4.023;
   1:  PR[GP1:91,2] = PR[GP1:90,2] + -1.796;
   1:L PR[91] R[100]mm/sec CNT100;
   1:  PR[GP1:91,1] = PR[GP1:90,1] + -0.454;
   1:  PR[GP1:91,2] = PR[GP1:90,2] + -0.472;
   1:L PR[91] R[100]mm/sec CNT100;
   1:  PR[GP1:91,1] = PR[GP1:90,1] + 0.667;
   1:L PR[91] R[100]mm/sec CNT100;
   1:  PR[GP1:91,1] = PR[GP1:90,1] + 4.236;
   1:  PR[GP1:91,2] = PR[GP1:90,2] + -1.796;
   1:L PR[91] R[100]mm/sec CNT100;
   1:  PR[GP1:91,1] = PR[GP1:90,1] + 6.052;
   1:  PR[GP1:91,2] = PR[GP1:90,2] + -5.076;
   1:L PR[91] R[100]mm/sec CNT100;
   1:  PR[GP1:91,1] = PR[GP1:90,1] + 8.085;
   1:  PR[GP1:91,2] = PR[GP1:90,2] + -10.871;
   1:L PR[91] R[100]mm/sec CNT100;
   1:  PR[GP1:91,1] = PR[GP1:90,1] + 8.921;
   1:  PR[GP1:91,2] = PR[GP1:90,2] + -14.227;
   1:L PR[91] R[100]mm/sec CNT100;
   1:  PR[GP1:91,1] = PR[GP1:90,1] + 10.319;
   1:  PR[GP1:91,2] = PR[GP1:90,2] + -17.267;
   1:L PR[91] R[100]mm/sec CNT100;
   1:  PR[GP1:91,1] = PR[GP1:90,1] + 14.243;
   1:  PR[GP1:91,2] = PR[GP1:90,2] + -21.821;
   1:L PR[91] R[100]mm/sec CNT100;
   1:  PR[GP1:91,1] = PR[GP1:90,1] + 16.246;
   1:  PR[GP1:91,2] = PR[GP1:90,2] + -24.640;
   1:L PR[91] R[100]mm/sec CNT100;
   1:  PR[GP1:91,1] = PR[GP1:90,1] + 18.658;
   1:  PR[GP1:91,2] = PR[GP1:90,2] + -26.960;
   1:L PR[91] R[100]mm/sec CNT100;
   1:  PR[GP1:91,1] = PR[GP1:90,1] + 23.971;
   1:  PR[GP1:91,2] = PR[GP1:90,2] + -29.764;
   1:L PR[91] R[100]mm/sec CNT100;
   1:  PR[GP1:91,1] = PR[GP1:90,1] + 26.866;
   1:  PR[GP1:91,2] = PR[GP1:90,2] + -31.657;
   1:L PR[91] R[100]mm/sec CNT100;
   1:  PR[GP1:91,1] = PR[GP1:90,1] + 29.958;
   1:  PR[GP1:91,2] = PR[GP1:90,2] + -32.935;
   1:L PR[91] R[100]mm/sec CNT100;
   1:  PR[GP1:91,1] = PR[GP1:90,1] + 35.931;
   1:  PR[GP1:91,2] = PR[GP1:90,2] + -33.606;
   1:L PR[91] R[100]mm/sec CNT100;
   1:  PR[GP1:91,1] = PR[GP1:90,1] + 39.317;
   1:  PR[GP1:91,2] = PR[GP1:90,2] + -34.311;
   1:L PR[91] R[100]mm/sec CNT100;
   1:  PR[GP1:91,1] = PR[GP1:90,1] + 42.663;
   1:  PR[GP1:91,2] = PR[GP1:90,2] + -34.371;
   1:L PR[91] R[100]mm/sec CNT100;
   1:  PR[GP1:91,1] = PR[GP1:90,1] + 48.468;
   1:  PR[GP1:91,2] = PR[GP1:90,2] + -32.814;
   1:L PR[91] R[100]mm/sec CNT100;
   1:  PR[GP1:91,1] = PR[GP1:90,1] + 51.877;
   1:  PR[GP1:91,2] = PR[GP1:90,2] + -32.233;
   1:L PR[91] R[100]mm/sec CNT100;
   1:  PR[GP1:91,1] = PR[GP1:90,1] + 55.014;
   1:  PR[GP1:91,2] = PR[GP1:90,2] + -31.068;
   1:L PR[91] R[100]mm/sec CNT100;
   1:  PR[GP1:91,1] = PR[GP1:90,1] + 59.847;
   1:  PR[GP1:91,2] = PR[GP1:90,2] + -27.500;
   1:L PR[91] R[100]mm/sec CNT100;
   1:  PR[GP1:91,1] = PR[GP1:90,1] + 62.809;
   1:  PR[GP1:91,2] = PR[GP1:90,2] + -25.714;
   1:L PR[91] R[100]mm/sec CNT100;
   1:  PR[GP1:91,1] = PR[GP1:90,1] + 65.304;
   1:  PR[GP1:91,2] = PR[GP1:90,2] + -23.483;
   1:L PR[91] R[100]mm/sec CNT100;
   1:  PR[GP1:91,1] = PR[GP1:90,1] + 68.502;
   1:  PR[GP1:91,2] = PR[GP1:90,2] + -18.393;
   1:L PR[91] R[100]mm/sec CNT100;
   1:  PR[GP1:91,1] = PR[GP1:90,1] + 70.607;
   1:  PR[GP1:91,2] = PR[GP1:90,2] + -15.648;
   1:L PR[91] R[100]mm/sec CNT100;
   1:  PR[GP1:91,1] = PR[GP1:90,1] + 72.114;
   1:  PR[GP1:91,2] = PR[GP1:90,2] + -12.661;
   1:L PR[91] R[100]mm/sec CNT100;
   1:  PR[GP1:91,1] = PR[GP1:90,1] + 73.232;
   1:  PR[GP1:91,2] = PR[GP1:90,2] + -6.756;
   1:L PR[91] R[100]mm/sec CNT100;
   1:  PR[GP1:91,1] = PR[GP1:90,1] + 74.189;
   1:  PR[GP1:91,2] = PR[GP1:90,2] + -3.432;
   1:L PR[91] R[100]mm/sec CNT100;
   1:  PR[GP1:91,1] = PR[GP1:90,1] + 74.501;
   1:  PR[GP1:91,2] = PR[GP1:90,2] + -0.100;
   1:L PR[91] R[100]mm/sec CNT100;
   1:  PR[GP1:91,1] = PR[GP1:90,1] + 73.384;
   1:  PR[GP1:91,2] = PR[GP1:90,2] + 5.805;
   1:L PR[91] R[100]mm/sec CNT100;
   1:  PR[GP1:91,1] = PR[GP1:90,1] + 73.061;
   1:  PR[GP1:91,2] = PR[GP1:90,2] + 9.249;
   1:L PR[91] R[100]mm/sec CNT100;
   1:  PR[GP1:91,1] = PR[GP1:90,1] + 72.127;
   1:  PR[GP1:91,2] = PR[GP1:90,2] + 12.492;
   1:L PR[91] R[100]mm/sec CNT100;
   1:  PR[GP1:91,1] = PR[GP1:90,1] + 70.594;
   1:  PR[GP1:91,2] = PR[GP1:90,2] + 15.529;
   1:L PR[91] R[100]mm/sec CNT100;
   1:  PR[GP1:91,1] = PR[GP1:90,1] + 67.396;
   1:  PR[GP1:91,2] = PR[GP1:90,2] + 20.620;
   1:L PR[91] R[100]mm/sec CNT100;
   1:  PR[GP1:91,1] = PR[GP1:90,1] + 65.325;
   1:  PR[GP1:91,2] = PR[GP1:90,2] + 23.320;
   1:L PR[91] R[100]mm/sec CNT100;
   1:  PR[GP1:91,1] = PR[GP1:90,1] + 62.788;
   1:  PR[GP1:91,2] = PR[GP1:90,2] + 25.588;
   1:L PR[91] R[100]mm/sec CNT100;
   1:  PR[GP1:91,1] = PR[GP1:90,1] + 57.955;
   1:  PR[GP1:91,2] = PR[GP1:90,2] + 29.157;
   1:L PR[91] R[100]mm/sec CNT100;
   1:  PR[GP1:91,1] = PR[GP1:90,1] + 55.041;
   1:  PR[GP1:91,2] = PR[GP1:90,2] + 30.914;
   1:L PR[91] R[100]mm/sec CNT100;
   1:  PR[GP1:91,1] = PR[GP1:90,1] + 51.851;
   1:  PR[GP1:91,2] = PR[GP1:90,2] + 32.099;
   1:L PR[91] R[100]mm/sec CNT100;
   1:  PR[GP1:91,1] = PR[GP1:90,1] + 46.046;
   1:  PR[GP1:91,2] = PR[GP1:90,2] + 33.656;
   1:L PR[91] R[100]mm/sec CNT100;
   1:  PR[GP1:91,1] = PR[GP1:90,1] + 42.691;
   1:  PR[GP1:91,2] = PR[GP1:90,2] + 34.228;
   1:L PR[91] R[100]mm/sec CNT100;
   1:  PR[GP1:91,1] = PR[GP1:90,1] + 39.289;
   1:  PR[GP1:91,2] = PR[GP1:90,2] + 34.166;
   1:L PR[91] R[100]mm/sec CNT100;
   1:  PR[GP1:91,1] = PR[GP1:90,1] + 33.316;
   1:  PR[GP1:91,2] = PR[GP1:90,2] + 33.495;
   1:L PR[91] R[100]mm/sec CNT100;
   1:  PR[GP1:91,1] = PR[GP1:90,1] + 29.984;
   1:  PR[GP1:91,2] = PR[GP1:90,2] + 32.802;
   1:L PR[91] R[100]mm/sec CNT100;
   1:  PR[GP1:91,1] = PR[GP1:90,1] + 26.840;
   1:  PR[GP1:91,2] = PR[GP1:90,2] + 31.502;
   1:L PR[91] R[100]mm/sec CNT100;
   1:  PR[GP1:91,1] = PR[GP1:90,1] + 21.527;
   1:  PR[GP1:91,2] = PR[GP1:90,2] + 28.698;
   1:L PR[91] R[100]mm/sec CNT100;
   1:  PR[GP1:91,1] = PR[GP1:90,1] + 18.679;
   1:  PR[GP1:91,2] = PR[GP1:90,2] + 26.835;
   1:L PR[91] R[100]mm/sec CNT100;
   1:  PR[GP1:91,1] = PR[GP1:90,1] + 16.226;
   1:  PR[GP1:91,2] = PR[GP1:90,2] + 24.477;
   1:L PR[91] R[100]mm/sec CNT100;
   1:  PR[GP1:91,1] = PR[GP1:90,1] + 12.302;
   1:  PR[GP1:91,2] = PR[GP1:90,2] + 19.923;
   1:L PR[91] R[100]mm/sec CNT100;
   1:  PR[GP1:91,1] = PR[GP1:90,1] + 10.331;
   1:  PR[GP1:91,2] = PR[GP1:90,2] + 17.149;
   1:L PR[91] R[100]mm/sec CNT100;
   1:  PR[GP1:91,1] = PR[GP1:90,1] + 8.909;
   1:  PR[GP1:91,2] = PR[GP1:90,2] + 14.058;
   1:L PR[91] R[100]mm/sec CNT100;
   1:  PR[GP1:91,1] = PR[GP1:90,1] + 6.921;
   1:  PR[GP1:91,2] = PR[GP1:90,2] + 8.390;
   1:L PR[91] R[100]mm/sec CNT100;
   1:  PR[GP1:91,1] = PR[GP1:90,1] + 6.066;
   1:  PR[GP1:91,2] = PR[GP1:90,2] + 4.956;
   1:L PR[91] R[100]mm/sec CNT100;
   1:  PR[GP1:91,1] = PR[GP1:90,1] + 4.236;
   1:  PR[GP1:91,2] = PR[GP1:90,2] + 1.652;
   1:L PR[91] R[100]mm/sec CNT100;
   1:  PR[GP1:91,1] = PR[GP1:90,1] + 0.667;
   1:  PR[GP1:91,2] = PR[GP1:90,2] + 0.328;
   1:L PR[91] R[100]mm/sec CNT100;
   1:  PR[GP1:91,1] = PR[GP1:90,1] + -0.454;
   1:L PR[91] R[100]mm/sec CNT100;
   1:  ! -- Layer/Ebene 8 -- !;
   1:  PR[91] = PR[90];
   1:  PR[GP1:91,1] = PR[GP1:90,1] + -4.023;
   1:  PR[GP1:91,2] = PR[GP1:90,2] + 1.652;
   1:  PR[GP1:91,3] = PR[GP1:90,3] + 5.185;
   1:L PR[91] R[100]mm/sec CNT100;
   1:  PR[GP1:91,1] = PR[GP1:90,1] + -5.839;
   1:  PR[GP1:91,2] = PR[GP1:90,2] + 4.932;
   1:L PR[91] R[100]mm/sec CNT100;
   1:  PR[GP1:91,1] = PR[GP1:90,1] + -7.544;
   1:  PR[GP1:91,2] = PR[GP1:90,2] + 9.791;
   1:L PR[91] R[100]mm/sec CNT100;
   1:  PR[GP1:91,1] = PR[GP1:90,1] + -8.500;
   1:  PR[GP1:91,2] = PR[GP1:90,2] + 13.631;
   1:L PR[91] R[100]mm/sec CNT100;
   1:  PR[GP1:91,1] = PR[GP1:90,1] + -10.106;
   1:  PR[GP1:91,2] = PR[GP1:90,2] + 17.124;
   1:L PR[91] R[100]mm/sec CNT100;
   1:  PR[GP1:91,1] = PR[GP1:90,1] + -13.382;
   1:  PR[GP1:91,2] = PR[GP1:90,2] + 20.926;
   1:L PR[91] R[100]mm/sec CNT100;
   1:  PR[GP1:91,1] = PR[GP1:90,1] + -15.674;
   1:  PR[GP1:91,2] = PR[GP1:90,2] + 24.151;
   1:L PR[91] R[100]mm/sec CNT100;
   1:  PR[GP1:91,1] = PR[GP1:90,1] + -18.445;
   1:  PR[GP1:91,2] = PR[GP1:90,2] + 26.816;
   1:L PR[91] R[100]mm/sec CNT100;
   1:  PR[GP1:91,1] = PR[GP1:90,1] + -22.881;
   1:  PR[GP1:91,2] = PR[GP1:90,2] + 29.157;
   1:L PR[91] R[100]mm/sec CNT100;
   1:  PR[GP1:91,1] = PR[GP1:90,1] + -26.193;
   1:  PR[GP1:91,2] = PR[GP1:90,2] + 31.323;
   1:L PR[91] R[100]mm/sec CNT100;
   1:  PR[GP1:91,1] = PR[GP1:90,1] + -29.745;
   1:  PR[GP1:91,2] = PR[GP1:90,2] + 32.792;
   1:L PR[91] R[100]mm/sec CNT100;
   1:  PR[GP1:91,1] = PR[GP1:90,1] + -34.732;
   1:  PR[GP1:91,2] = PR[GP1:90,2] + 33.351;
   1:L PR[91] R[100]mm/sec CNT100;
   1:  PR[GP1:91,1] = PR[GP1:90,1] + -38.606;
   1:  PR[GP1:91,2] = PR[GP1:90,2] + 34.157;
   1:L PR[91] R[100]mm/sec CNT100;
   1:  PR[GP1:91,1] = PR[GP1:90,1] + -42.450;
   1:  PR[GP1:91,2] = PR[GP1:90,2] + 34.227;
   1:L PR[91] R[100]mm/sec CNT100;
   1:  PR[GP1:91,1] = PR[GP1:90,1] + -47.297;
   1:  PR[GP1:91,2] = PR[GP1:90,2] + 32.927;
   1:L PR[91] R[100]mm/sec CNT100;
   1:  PR[GP1:91,1] = PR[GP1:90,1] + -51.197;
   1:  PR[GP1:91,2] = PR[GP1:90,2] + 32.263;
   1:L PR[91] R[100]mm/sec CNT100;
   1:  PR[GP1:91,1] = PR[GP1:90,1] + -54.801;
   1:  PR[GP1:91,2] = PR[GP1:90,2] + 30.924;
   1:L PR[91] R[100]mm/sec CNT100;
   1:  PR[GP1:91,1] = PR[GP1:90,1] + -58.836;
   1:  PR[GP1:91,2] = PR[GP1:90,2] + 27.945;
   1:L PR[91] R[100]mm/sec CNT100;
   1:  PR[GP1:91,1] = PR[GP1:90,1] + -62.225;
   1:  PR[GP1:91,2] = PR[GP1:90,2] + 25.901;
   1:L PR[91] R[100]mm/sec CNT100;
   1:  PR[GP1:91,1] = PR[GP1:90,1] + -65.091;
   1:  PR[GP1:91,2] = PR[GP1:90,2] + 23.339;
   1:L PR[91] R[100]mm/sec CNT100;
   1:  PR[GP1:91,1] = PR[GP1:90,1] + -67.761;
   1:  PR[GP1:91,2] = PR[GP1:90,2] + 19.089;
   1:L PR[91] R[100]mm/sec CNT100;
   1:  PR[GP1:91,1] = PR[GP1:90,1] + -70.169;
   1:  PR[GP1:91,2] = PR[GP1:90,2] + 15.949;
   1:L PR[91] R[100]mm/sec CNT100;
   1:  PR[GP1:91,1] = PR[GP1:90,1] + -71.901;
   1:  PR[GP1:91,2] = PR[GP1:90,2] + 12.517;
   1:L PR[91] R[100]mm/sec CNT100;
   1:  PR[GP1:91,1] = PR[GP1:90,1] + -72.834;
   1:  PR[GP1:91,2] = PR[GP1:90,2] + 7.586;
   1:L PR[91] R[100]mm/sec CNT100;
   1:  PR[GP1:91,1] = PR[GP1:90,1] + -73.929;
   1:  PR[GP1:91,2] = PR[GP1:90,2] + 3.784;
   1:L PR[91] R[100]mm/sec CNT100;
   1:  PR[GP1:91,1] = PR[GP1:90,1] + -74.288;
   1:  PR[GP1:91,2] = PR[GP1:90,2] + -0.044;
   1:L PR[91] R[100]mm/sec CNT100;
   1:  PR[GP1:91,1] = PR[GP1:90,1] + -73.355;
   1:  PR[GP1:91,2] = PR[GP1:90,2] + -4.974;
   1:L PR[91] R[100]mm/sec CNT100;
   1:  PR[GP1:91,1] = PR[GP1:90,1] + -72.986;
   1:  PR[GP1:91,2] = PR[GP1:90,2] + -8.914;
   1:L PR[91] R[100]mm/sec CNT100;
   1:  PR[GP1:91,1] = PR[GP1:90,1] + -71.914;
   1:  PR[GP1:91,2] = PR[GP1:90,2] + -12.635;
   1:L PR[91] R[100]mm/sec CNT100;
   1:  PR[GP1:91,1] = PR[GP1:90,1] + -70.157;
   1:  PR[GP1:91,2] = PR[GP1:90,2] + -16.118;
   1:L PR[91] R[100]mm/sec CNT100;
   1:  PR[GP1:91,1] = PR[GP1:90,1] + -67.486;
   1:  PR[GP1:91,2] = PR[GP1:90,2] + -20.369;
   1:L PR[91] R[100]mm/sec CNT100;
   1:  PR[GP1:91,1] = PR[GP1:90,1] + -65.112;
   1:  PR[GP1:91,2] = PR[GP1:90,2] + -23.464;
   1:L PR[91] R[100]mm/sec CNT100;
   1:  PR[GP1:91,1] = PR[GP1:90,1] + -62.204;
   1:  PR[GP1:91,2] = PR[GP1:90,2] + -26.064;
   1:L PR[91] R[100]mm/sec CNT100;
   1:  PR[GP1:91,1] = PR[GP1:90,1] + -58.168;
   1:  PR[GP1:91,2] = PR[GP1:90,2] + -29.044;
   1:L PR[91] R[100]mm/sec CNT100;
   1:  PR[GP1:91,1] = PR[GP1:90,1] + -54.828;
   1:  PR[GP1:91,2] = PR[GP1:90,2] + -31.058;
   1:L PR[91] R[100]mm/sec CNT100;
   1:  PR[GP1:91,1] = PR[GP1:90,1] + -51.171;
   1:  PR[GP1:91,2] = PR[GP1:90,2] + -32.417;
   1:L PR[91] R[100]mm/sec CNT100;
   1:  PR[GP1:91,1] = PR[GP1:90,1] + -46.324;
   1:  PR[GP1:91,2] = PR[GP1:90,2] + -33.717;
   1:L PR[91] R[100]mm/sec CNT100;
   1:  PR[GP1:91,1] = PR[GP1:90,1] + -42.478;
   1:  PR[GP1:91,2] = PR[GP1:90,2] + -34.372;
   1:L PR[91] R[100]mm/sec CNT100;
   1:  PR[GP1:91,1] = PR[GP1:90,1] + -38.578;
   1:  PR[GP1:91,2] = PR[GP1:90,2] + -34.301;
   1:L PR[91] R[100]mm/sec CNT100;
   1:  PR[GP1:91,1] = PR[GP1:90,1] + -33.591;
   1:  PR[GP1:91,2] = PR[GP1:90,2] + -33.741;
   1:L PR[91] R[100]mm/sec CNT100;
   1:  PR[GP1:91,1] = PR[GP1:90,1] + -29.772;
   1:  PR[GP1:91,2] = PR[GP1:90,2] + -32.946;
   1:L PR[91] R[100]mm/sec CNT100;
   1:  PR[GP1:91,1] = PR[GP1:90,1] + -26.167;
   1:  PR[GP1:91,2] = PR[GP1:90,2] + -31.456;
   1:L PR[91] R[100]mm/sec CNT100;
   1:  PR[GP1:91,1] = PR[GP1:90,1] + -21.731;
   1:  PR[GP1:91,2] = PR[GP1:90,2] + -29.114;
   1:L PR[91] R[100]mm/sec CNT100;
   1:  PR[GP1:91,1] = PR[GP1:90,1] + -18.466;
   1:  PR[GP1:91,2] = PR[GP1:90,2] + -26.980;
   1:L PR[91] R[100]mm/sec CNT100;
   1:  PR[GP1:91,1] = PR[GP1:90,1] + -15.654;
   1:  PR[GP1:91,2] = PR[GP1:90,2] + -24.275;
   1:L PR[91] R[100]mm/sec CNT100;
   1:  PR[GP1:91,1] = PR[GP1:90,1] + -12.378;
   1:  PR[GP1:91,2] = PR[GP1:90,2] + -20.473;
   1:L PR[91] R[100]mm/sec CNT100;
   1:  PR[GP1:91,1] = PR[GP1:90,1] + -10.118;
   1:  PR[GP1:91,2] = PR[GP1:90,2] + -17.294;
   1:L PR[91] R[100]mm/sec CNT100;
   1:  PR[GP1:91,1] = PR[GP1:90,1] + -8.488;
